(* IEC 61131-3 sources: SmartHomeNew/snapshots/clean_build_2026_04_15, 37 files *)

(* ---- E_Debug_Log_Level.dut ---- *)
{attribute 'strict'}
TYPE E_Debug_Log_Level :
(
    LOG_LEVEL_MINIMAL := 0,
    LOG_LEVEL_NORMAL := 1,
    LOG_LEVEL_VERBOSE := 2,
    LOG_LEVEL_DEBUG := 3
) USINT;
END_TYPE

(* ---- E_Zone_Access_Level.dut ---- *)
{attribute 'strict'}
TYPE E_Zone_Access_Level :
(
    ZONE_ACCESS_NONE := 0,
    ZONE_ACCESS_VIEW := 1,
    ZONE_ACCESS_CONTROL := 2,
    ZONE_ACCESS_CONFIG := 3,
    ZONE_ACCESS_FULL := 4
) USINT;
END_TYPE

(* ---- ST_BlackBox_Snapshot_V2.dut ---- *)
TYPE ST_BlackBox_Snapshot_V2 : STRUCT
    Gas_Alarm : BOOL;
    Fire_Alarm : BOOL;
    Flood_Alarm : BOOL;
    First_Fault_Type : BYTE;
    First_Fault_Source : BYTE;
END_STRUCT
END_TYPE

(* ---- ST_Boiler_Status.dut ---- *)
{attribute 'pack_mode' := '1'}
TYPE ST_Boiler_Status :
STRUCT
    Active : BOOL;
    Running : BOOL;
    Warning : BOOL;
    Error : BOOL;
    Error_ID : WORD;
    Power_Percent : REAL;
    Current_Power : REAL;
    Work_Seconds : UDINT;
    Work_Hours : REAL;
    Resource_Percent : REAL := 100.0;
    Last_Start : DT;
END_STRUCT
END_TYPE

(* ---- ST_Component_Maintenance.dut ---- *)
{attribute 'pack_mode' := '1'}
TYPE ST_Component_Maintenance :
STRUCT
    Is_Faulty : BOOL;
    Is_In_Maintenance : BOOL;
    Fallback_Value : REAL;
    Use_Last_Good_Value : BOOL;
END_STRUCT
END_TYPE

(* ---- ST_History_Event_V2.dut ---- *)
TYPE ST_History_Event_V2 : STRUCT
    Event_Code : UINT;
    Event_Value : REAL;
END_STRUCT
END_TYPE

(* ---- ST_Outdoor_Zone_Config.dut ---- *)
{attribute 'pack_mode' := '1'}
TYPE ST_Outdoor_Zone_Config :
STRUCT
    zone_id : BYTE := 0;
    lighting_circuit_id : BYTE := 0;
    auto_enabled : BOOL := TRUE;
    party_mode_enabled : BOOL := FALSE;
END_STRUCT
END_TYPE

(* ---- ST_Rule_Action.dut ---- *)
{attribute 'pack_mode' := '1'}
TYPE ST_Rule_Action :
STRUCT
    Active : BOOL;
    Triggered : BOOL;
    Action_Type : E_Rule_Action_Type;
    Target_ID : BYTE;
    Value : REAL;
END_STRUCT
END_TYPE

(* ---- ST_Valve_Test_Config.dut ---- *)
{attribute 'pack_mode' := '1'}
TYPE ST_Valve_Test_Config :
STRUCT
    valve_id : BYTE := 0;
    test_interval_days : UDINT := 7;
    Nominal_Current : REAL := 0.5;
    nominal_close_time_sec : REAL := 10.0;
    enabled : BOOL := TRUE;
END_STRUCT
END_TYPE

(* ---- GVL_COMMAND.gvl ---- *)
{attribute 'qualified_only'}
VAR_GLOBAL
    G_Gas_Valve_Close : BOOL := FALSE; // Команда: Закрыть газовый клапан
    G_Boiler_Stop : BOOL := FALSE; // Команда: Остановка котлов
    G_Supply_100_Req : BOOL := FALSE; // Команда: Приток 100%
    G_Supply_80_Req : BOOL := FALSE; // Команда: Приток 80%
    G_Vent_PV3_Boost : BOOL := FALSE; // Команда: Форсированный режим ПВ-3
    G_Exhaust_100_Req : BOOL := FALSE; // Команда: Вытяжка 100%
    G_Vent_Stop : BOOL := FALSE; // Команда: Остановка вентиляции
    G_Close_Valve_35 : BOOL := FALSE; // Команда: Закрыть вводной кран 1
    G_Close_Valve_36 : BOOL := FALSE; // Команда: Закрыть вводной кран 2
    G_Gate_Open : BOOL;
    G_Wicket_Open : BOOL;
    G_Lock_1_Open : BOOL;
    G_Lock_1_Close : BOOL;
    G_Lock_2_Open : BOOL;
    G_Lock_2_Close : BOOL;
    G_Reset_Errors : BOOL := FALSE; // Команда: Сброс ошибок
    G_Scenario_Request : E_SCENARIO_TYPE := E_SCENARIO_TYPE.SCENARIO_NONE; // Запрос на активацию сценария

    // Команды от шлюза
    G_Arm_Req : BOOL;
    G_Disarm_Req : BOOL;
    G_PIN_Code : STRING(4);
    G_RFID_Tag : STRING(20);
    G_2FA_Code_In : STRING(6);
    G_Send_2FA_Req : BOOL;
    G_2FA_Code_Out : STRING(6);
    G_Lighting_Override : ARRAY[1..32] OF BYTE;
    G_Blinds_Override : ARRAY[1..GVL_CONSTANTS.C_MAX_BLINDS] OF BYTE;
    G_Socket_Override : ARRAY[1..GVL_CONSTANTS.C_MAX_SOCKETS] OF BOOL;
    CMD_Set_Manifold_Pump_In_Service : ARRAY[1..GVL_CONSTANTS.C_MAX_MANIFOLDS] OF BOOL;
    CMD_Set_DHW_Heating_Pump_In_Service : BOOL;
    CMD_Set_DHW_Circ_Pump_In_Service : BOOL;
    CMD_Dangerous_Action_Confirm : BOOL;
    CMD_Dangerous_Action_Request : BOOL;
    CMD_User_Access_Level : INT := 0;
    CMD_Valve_Test_Open : BOOL;
    CMD_Valve_Test_Close : BOOL;
    CMD_Valve_Test_Confirm : BOOL;
    CMD_Water_Valve_Test_Open : BOOL;
    CMD_Water_Valve_Test_Close : BOOL;
    CMD_Water_Valve_Test_Confirm : BOOL;
    CMD_Gas_Valve_Test_Open : BOOL;
    CMD_Gas_Valve_Test_Close : BOOL;
    CMD_Gas_Valve_Test_Confirm : BOOL;
    CMD_Water_Selective_Recover : BOOL;
    CMD_Gas_Selective_Recover : BOOL;
END_VAR

(* ---- GVL_CONSTANTS.gvl ---- *)
{attribute 'qualified_only'}
VAR_GLOBAL CONSTANT
    // Размеры массивов (конфигурация системы)
    C_MAX_ZONES            : INT := 16; // Максимальное количество зон (комнат)
    C_MAX_LIGHTING_ZONES   : INT := 32; // Алиас для контуров освещения
    C_MAX_HEATING_CIRCUITS : INT := 8;  // Алиас для контуров отопления
    C_MAX_CLIMATE_ZONES    : INT := 16; // Алиас для климатических зон
    C_MAX_LIGHT_ZONES      : INT := 32; // Алиас для световых зон
    C_MAX_SOCKETS          : INT := 36; // Максимальное количество управляемых розеток
    C_MAX_BLINDS           : INT := 20; // Максимальное количество штор/жалюзи
    C_MAX_ALARMS           : INT := 20; // Максимальное количество активных тревог
    C_MAX_RULES            : INT := 20; // Максимальное количество правил (движок правил)
    C_MAX_MANIFOLDS        : INT := 5;  // Максимальное количество коллекторов
    C_MAX_BOILERS          : INT := 2;  // Максимальное количество котлов
    C_MAX_SUPPLY_FANS      : INT := 3;  // Максимальное количество приточных вентиляторов
    C_MAX_EXHAUST_FANS     : INT := 5;  // Максимальное количество вытяжных вентиляторов
    C_MAX_SECURITY_SENSORS : INT := 15; // Максимальное количество датчиков безопасности (герконы, стекло)
    C_MAX_FLOOD_SENSORS    : INT := 12; // Максимальное количество датчиков протечки
    C_MAX_DOOR_SENSORS     : INT := 8;  // Максимальное количество датчиков дверей
    C_MAX_CO_SENSORS       : INT := 8;  // Максимальное количество датчиков CO
    C_MAX_METHANE_SENSORS  : INT := 2;  // Максимальное количество датчиков метана
    C_MAX_VENT_UNITS       : INT := 8;  // Максимальное количество вентустановок
    C_MAX_SUPPLY_TEMPS     : INT := 2;  // Максимальное количество датчиков температуры притока
    C_MAX_SMOKE_SENSORS    : INT := 6;  // Максимальное количество датчиков дыма
    C_MAX_SCENARIOS        : INT := 6;  // Максимальное количество сценариев
    C_MAX_OUTDOOR_ZONES    : INT := 4;  // Максимальное количество зон уличного освещения
    C_MAX_ACCESS_CODES     : INT := 10; // Максимальное количество кодов доступа
    C_MAX_WET_ZONES        : INT := 4;  // Максимальное количество "мокрых" зон (санузлы)
    C_MAX_CALIBRATIONS     : INT := 20; // Максимальное количество калибровок датчиков
    C_MAX_MODULES          : INT := 10; // Максимальное количество модулей ввода-вывода
    C_MAX_CLEANING_MODES   : INT := 3;  // Максимальное количество режимов уборки
    C_MAX_ALLOWED_IPS      : INT := 5;  // Максимальное количество разрешенных IP-адресов
    C_MAX_VENT_SUPPLY_MODES: INT := 3;  // Максимальное количество режимов притока вентиляции
    C_MAX_SECURITY_PHONES  : INT := 5;  // Максимальное количество телефонов для оповещения
    C_MAX_FLOOD_VALVES     : INT := 3;  // Максимальное количество кранов защиты от протечек
    C_MAX_HUMIDITY_SENSORS : INT := 8;  // Максимальное количество датчиков влажности
    C_MAX_CO2_SENSORS      : INT := 8;  // Максимальное количество датчиков CO2
    C_MAX_CIRCUITS_PER_MANIFOLD : INT := 4; // Максимальное количество контуров на коллектор
    C_MAX_TREND_DATA_POINTS: INT := 100; // Максимальное количество точек данных для трендов
    C_MAX_HISTORY_RECORDS  : INT := 100; // Максимальное количество записей в истории
    C_MAX_DEBUG_LOGS       : INT := 1000; // Максимальное количество записей в логе отладки
    C_MAX_GATEWAY_COMMANDS : INT := 10; // Максимальное количество команд в буфере шлюза
    C_MAX_STATE_SNAPSHOTS  : INT := 10; // Максимальное количество снимков состояния
    C_MAX_BLACKBOX_RECORDS : INT := 100; // Максимальное количество записей черного ящика
    C_MAX_PRESENCE_HISTORY : INT := 1008; // Максимальное количество записей истории присутствия
    C_MAX_MODBUS_REGISTERS : INT := 201; // Максимальное количество регистров Modbus
    C_MAX_DEDUPLICATION_HISTORY : INT := 100; // Максимальное количество записей истории дедупликации
    C_MAX_NVRAM_RECORDS    : INT := 100; // Максимальное количество записей NVRAM
    C_MAX_NVRAM_DATA       : INT := 128; // Максимальный размер данных NVRAM

    // Аналоговые входы (4-20mA, 0-10V)
    C_ANALOG_RAW_MAX       : WORD := 27648; // Максимальное значение АЦП (100%)
    C_ANALOG_4MA_RAW       : WORD := 5529;  // Значение АЦП для 4mA (20% от 27648)
    C_ANALOG_3_6MA_RAW     : WORD := 4976;  // Порог обрыва NAMUR NE43 (< 3.6mA)
    C_ANALOG_21MA_RAW      : WORD := 29030; // Порог КЗ NAMUR NE43 (> 21mA)
    C_ANALOG_10V_MAX_RAW   : WORD := 30000; // Порог выхода за пределы 0-10V

    // Временные константы (в миллисекундах)
    C_MS_IN_SECOND         : UDINT := 1000;
    C_MS_IN_MINUTE         : UDINT := 60000;
    C_MS_IN_HOUR           : UDINT := 3600000;
    C_MS_IN_DAY            : UDINT := 86400000;

    // Пороги мощности для каскада котлов (0..500%)
    C_BOILER_CASCADE_MIN_DEMAND : REAL := 25.0; // Минимальный запрос для включения ведущего котла (5% от одного коллектора)
    C_BOILER_CASCADE_HIGH_DEMAND : REAL := 250.0; // Высокий запрос для включения второго котла (50% от общей мощности)
END_VAR

(* ---- GVL_GATEWAY.gvl ---- *)
{attribute 'qualified_only'}
VAR_GLOBAL
    G_Gateway_Command : ST_Gateway_Command;
    G_Gateway_Command_Received : BOOL;
    G_Gateway_Send_2FA : BOOL;
    G_Gateway_2FA_Code : STRING(6);
    G_Gateway_Telegram_Msg : STRING(200);
    G_Gateway_Send_Telegram : BOOL;
    G_Gateway_HMI_Status_Message : STRING(200);
    G_Gateway_Ping_OK : BOOL;
    G_Gateway_Data_Ready : BOOL;
    G_Gateway_Modbus_Registers : ARRAY[0..GVL_CONSTANTS.C_MAX_MODBUS_REGISTERS-1] OF WORD;
END_VAR

(* ---- GVL_STATE.gvl ---- *)
{attribute 'qualified_only'}
VAR_GLOBAL
    G_Floor_Temps : ARRAY[1..8] OF REAL; // Массив текущих температур поверхности пола
    G_Room_Temps : ARRAY[1..GVL_CONSTANTS.C_MAX_ZONES] OF REAL;
    G_Room_Hum : ARRAY[1..GVL_CONSTANTS.C_MAX_ZONES] OF REAL;
    G_Room_CO2 : ARRAY[1..GVL_CONSTANTS.C_MAX_ZONES] OF REAL;
    G_Motion_Sensors : ARRAY[1..32] OF BOOL;
    G_Door_Sensors : ARRAY[1..GVL_CONSTANTS.C_MAX_DOOR_SENSORS] OF BOOL;
    G_Window_Sensors : ARRAY[1..GVL_CONSTANTS.C_MAX_ZONES] OF BOOL;
    G_Water_Sensors : ARRAY[1..GVL_CONSTANTS.C_MAX_FLOOD_SENSORS] OF BOOL;
    G_Smoke_Sensors : ARRAY[1..GVL_CONSTANTS.C_MAX_SMOKE_SENSORS] OF BOOL;
    G_Methane_Sensors : ARRAY[1..GVL_CONSTANTS.C_MAX_METHANE_SENSORS] OF REAL;
    G_CO_Sensors : ARRAY[1..GVL_CONSTANTS.C_MAX_CO_SENSORS] OF REAL;
    G_Manifold_Pressures : ARRAY[1..GVL_CONSTANTS.C_MAX_MANIFOLDS] OF REAL;
    G_Manifold_Currents : ARRAY[1..GVL_CONSTANTS.C_MAX_MANIFOLDS] OF REAL;
    G_Manifold_T_Supply : ARRAY[1..GVL_CONSTANTS.C_MAX_MANIFOLDS] OF REAL;
    G_Manifold_T_Return : ARRAY[1..GVL_CONSTANTS.C_MAX_MANIFOLDS] OF REAL;
    G_Boiler_Flame : ARRAY[1..GVL_CONSTANTS.C_MAX_BOILERS] OF BOOL;
    G_Boiler_Error : ARRAY[1..GVL_CONSTANTS.C_MAX_BOILERS] OF BOOL;
    G_Boiler_OT_Online : ARRAY[1..GVL_CONSTANTS.C_MAX_BOILERS] OF BOOL; // Статус доступности OpenTherm-канала котла от реального OT-адаптера/драйвера
    G_Boiler_OT_Enable : ARRAY[1..GVL_CONSTANTS.C_MAX_BOILERS] OF BOOL; // Команды разрешения через OpenTherm
    G_Boiler_OT_Setpoint : ARRAY[1..GVL_CONSTANTS.C_MAX_BOILERS] OF REAL; // Уставки через OpenTherm
    G_Physical_Switches : ARRAY[1..32] OF BOOL;
    G_Socket_Switches : ARRAY[1..GVL_CONSTANTS.C_MAX_SOCKETS] OF BOOL; // Legacy-поле: локальные выключатели розеток не используются
    G_Outdoor_Temp : REAL;
    G_Supply_Temps : ARRAY[1..GVL_CONSTANTS.C_MAX_SUPPLY_TEMPS] OF REAL; // Температура приточного воздуха после калорифера
    G_DHW_Temp : REAL;
    G_DHW_Pressure : REAL;
    G_Zone_Valves : ARRAY[1..8] OF BOOL;
    G_Manifold_Pumps : ARRAY[1..GVL_CONSTANTS.C_MAX_MANIFOLDS] OF BOOL;
    G_Manifold_Valves : ARRAY[1..GVL_CONSTANTS.C_MAX_MANIFOLDS] OF REAL; // 0.0 - 1.0
    G_Manifold_End_Switches : ARRAY[1..GVL_CONSTANTS.C_MAX_MANIFOLDS] OF BOOL; // Концевики клапанов
    G_Supply_Fans : ARRAY[1..GVL_CONSTANTS.C_MAX_SUPPLY_FANS] OF REAL; // 0.0 - 1.0
    G_Exhaust_Fans : ARRAY[1..GVL_CONSTANTS.C_MAX_EXHAUST_FANS] OF REAL; // 0.0 - 1.0
    G_Vent_Heater_Power : ARRAY[1..GVL_CONSTANTS.C_MAX_BOILERS] OF REAL;
    G_Lighting_Levels : ARRAY[1..32] OF BYTE;
    G_Blinds_Positions : ARRAY[1..GVL_CONSTANTS.C_MAX_BLINDS] OF BYTE;
    G_Socket_States : ARRAY[1..GVL_CONSTANTS.C_MAX_SOCKETS] OF BOOL;
    G_DHW_Heating_Pump : BOOL;
    G_DHW_Circ_Pump : BOOL;
    G_Backup_Circulation_Pump : BOOL; // Резервный циркуляционный насос для антизамерзания при газовой аварии
    G_Electric_Heater_Enable : BOOL; // Сухой контакт электрического нагревателя для антизамерзания
    G_Safety_Gas_Alarm : BOOL;
    G_Safety_Leak_Alarm : BOOL;
    G_Safety_Smoke_Alarm : BOOL;
    G_Safety_Emergency_Stop : BOOL; // агрегированный аварийный стоп
    G_Safety_Gas_Latched : BOOL; // защёлкнутая газовая авария
    G_Safety_Leak_Latched : BOOL; // защёлкнутая авария протечки
    G_Safety_Smoke_Latched : BOOL; // защёлкнутая дымовая/пожарная авария
    G_Safety_Freeze_Risk : BOOL; // риск замерзания при защёлкнутой газовой аварии
    G_System_Mode : E_System_Operating_Mode := E_System_Operating_Mode.MODE_NORMAL; // Текущий режим работы системы
    G_System_Mode_Text : STRING(64);
    G_Heating_IO_Fault : BOOL;
    G_Heating_Sensor_Fault : BOOL;
    G_Heating_Subsystem_Degraded : BOOL;
    G_DHW_IO_Fault : BOOL;
    G_DHW_Sensor_Fault : BOOL;
    G_DHW_Subsystem_Degraded : BOOL;
    G_Ventilation_IO_Fault : BOOL;
    G_Ventilation_Subsystem_Degraded : BOOL;
    G_Lighting_IO_Fault : BOOL;
    G_Lighting_Subsystem_Degraded : BOOL;
    G_Access_Comm_Fault : BOOL;
    G_Evacuation_Lighting_Active : BOOL;
    G_Evac_Hazard_Zone : ARRAY[1..32] OF BOOL; // опасные зоны (дым/протечка)
    G_Evac_Guidance : ARRAY[1..32] OF INT; // -1 = избегать, 0 = нейтрально, +1 = к выходу
 // Активен режим световой эвакуации // Текстовый статус режима работы системы

    G_Rule_Actions : ARRAY[1..GVL_CONSTANTS.C_MAX_RULES] OF ST_Rule_Action;
    G_Sim_Lights : ARRAY[1..32] OF BOOL;
    G_Freeze_Hardware_Degraded : BOOL; // Деградация anti-freeze hardware
    G_Freeze_Hardware_Failed : BOOL; // Критический отказ anti-freeze hardware
    G_Water_Zone_Enable : ARRAY[1..32] OF BOOL; // Селективное открытие воды по зонам
    G_Water_Zone_Open_FB : ARRAY[1..32] OF BOOL; // Обратная связь: зональный клапан открыт
    G_Water_Zone_Close_FB : ARRAY[1..32] OF BOOL; // Обратная связь: зональный клапан закрыт
    G_Water_Zone_Exercise_Active : ARRAY[1..32] OF BOOL; // Профилактическая прокрутка шаровых кранов
END_VAR

(* ---- FB_Alarm_V2_Core.st ---- *)
FUNCTION_BLOCK FB_Alarm_V2_Core
VAR_INPUT
    VI_System_Time_MS : UDINT;
    VI_Pending_Alarms : ARRAY[1..10] OF ST_Alarm_Record;
END_VAR
VAR_IN_OUT
    VIO_Alarm_List : ARRAY[1..GVL_CONSTANTS.C_MAX_ALARMS] OF ST_Alarm_Record;
    VIO_Next_Alarm_ID : UDINT;
END_VAR
VAR_OUTPUT
    VO_Event_Pulse : BOOL;
    VO_Event_Code : UDINT;
    VO_Event_Value : REAL;
END_VAR

VO_Event_Pulse := FALSE;
VO_Event_Code := 0;
VO_Event_Value := 0.0;
END_FUNCTION_BLOCK

(* ---- FB_BlackBox_Recorder.st ---- *)
FUNCTION_BLOCK FB_BlackBox_Recorder
VAR_INPUT
    VI_Current_Data : ST_BlackBox_Record;
    VI_Freeze       : BOOL;
END_VAR
VAR_OUTPUT
    VO_Frozen       : BOOL;
    VO_Records_Count: INT;
END_VAR
VAR
    L_Write_Index   : INT := 0;
    L_Initialized   : BOOL := FALSE;
END_VAR

IF NOT L_Initialized THEN
    L_Write_Index := GVL_Retain.G_BlackBox_LastIndex;
    IF L_Write_Index < 0 OR L_Write_Index >= GVL_CONSTANTS.C_MAX_BLACKBOX_RECORDS THEN
        L_Write_Index := 0;
        GVL_Retain.G_BlackBox_LastIndex := 0;
    END_IF;
    L_Initialized := TRUE;
END_IF;

IF VI_Freeze THEN
    GVL_Retain.G_BlackBox_Frozen := TRUE;
END_IF;

VO_Frozen := GVL_Retain.G_BlackBox_Frozen;

IF NOT GVL_Retain.G_BlackBox_Frozen THEN
    GVL_Retain.G_BlackBox_Buffer[L_Write_Index] := VI_Current_Data;
    GVL_Retain.G_BlackBox_LastIndex := L_Write_Index;

    L_Write_Index := L_Write_Index + 1;
    IF L_Write_Index >= GVL_CONSTANTS.C_MAX_BLACKBOX_RECORDS THEN
        L_Write_Index := 0;
    END_IF;
END_IF;

VO_Records_Count := GVL_CONSTANTS.C_MAX_BLACKBOX_RECORDS; // Размер кольцевого буфера
// >>> BULK_SYNC_ANCHOR: FB_BlackBox_Recorder <<<

(* ---- FB_Boiler_Cascade_Manager.st ---- *)
FUNCTION_BLOCK FB_Boiler_Cascade_Manager
VAR_INPUT
    VI_Enable : BOOL;
    VI_System_Time_MS : UDINT;
    VI_Boiler_Stop : BOOL;

    VI_DHW_Heating_Demand : BOOL;
    VI_DHW_Target_Temp : REAL;

    VI_Target_Supply_Temp : REAL;
    VI_Demand_Power : REAL; // 0..500% (сумма запросов от 5 смесительных узлов)

    VI_Boiler_Flame_Status : ARRAY[1..GVL_CONSTANTS.C_MAX_BOILERS] OF BOOL;
    VI_Boiler_Error_Status : ARRAY[1..GVL_CONSTANTS.C_MAX_BOILERS] OF BOOL;
    VI_Boiler_OT_Online : ARRAY[1..GVL_CONSTANTS.C_MAX_BOILERS] OF BOOL;
    VI_Boiler_Modulation : ARRAY[1..GVL_CONSTANTS.C_MAX_BOILERS] OF REAL;
END_VAR

VAR_OUTPUT
    VO_Boiler_Enable : ARRAY[1..GVL_CONSTANTS.C_MAX_BOILERS] OF BOOL;
    VO_Boiler_Setpoint : ARRAY[1..GVL_CONSTANTS.C_MAX_BOILERS] OF REAL;
    VO_Lead_Boiler : BYTE;
END_VAR

VAR
    L_i : INT;
    L_Lead_Boiler : BYTE := 1;

    L_Last_Rotation_MS : UDINT := 0;
    L_Rotation_Initialized : BOOL := FALSE;
    L_Rotation_Period_MS : UDINT := 604800000; // 168h

    L_Lead_Available : BOOL;
    L_Reserve_Available : BOOL;
    L_Reserve_Boiler : BYTE;
    L_Start_Reserve : BOOL;
    L_Target_Setpoint : REAL;
    L_Flame_Miss_Timer : ARRAY[1..GVL_CONSTANTS.C_MAX_BOILERS] OF TON;
END_VAR

// Сброс выходов по умолчанию
FOR L_i := 1 TO GVL_CONSTANTS.C_MAX_BOILERS DO
    VO_Boiler_Enable[L_i] := FALSE;
    VO_Boiler_Setpoint[L_i] := 0.0;
END_FOR;

// Инициализация ротации
IF NOT L_Rotation_Initialized THEN
    L_Last_Rotation_MS := VI_System_Time_MS;
    L_Rotation_Initialized := TRUE;
END_IF;

// Принудительная остановка
IF VI_Boiler_Stop THEN
    VO_Lead_Boiler := L_Lead_Boiler;
    RETURN;
END_IF;

// Ротация строго каждые 168 часов
IF (VI_System_Time_MS - L_Last_Rotation_MS) >= L_Rotation_Period_MS THEN
    IF GVL_CONSTANTS.C_MAX_BOILERS > 1 THEN
        L_Lead_Boiler := 3 - L_Lead_Boiler;
    END_IF;
    L_Last_Rotation_MS := VI_System_Time_MS;
END_IF;

L_Reserve_Boiler := SEL(L_Lead_Boiler = 1, 1, 2);

L_Lead_Available :=
    VI_Boiler_OT_Online[L_Lead_Boiler] AND
    NOT VI_Boiler_Error_Status[L_Lead_Boiler];

L_Reserve_Available :=
    (GVL_CONSTANTS.C_MAX_BOILERS > 1) AND
    VI_Boiler_OT_Online[L_Reserve_Boiler] AND
    NOT VI_Boiler_Error_Status[L_Reserve_Boiler];

// Контроль "команда есть, пламени нет" для ведущего котла
L_Flame_Miss_Timer[L_Lead_Boiler](
    IN := VI_Enable AND L_Lead_Available AND NOT VI_DHW_Heating_Demand AND NOT VI_Boiler_Flame_Status[L_Lead_Boiler],
    PT := T#120s
);

IF L_Flame_Miss_Timer[L_Lead_Boiler].Q AND L_Reserve_Available THEN
    L_Lead_Boiler := L_Reserve_Boiler;
    L_Last_Rotation_MS := VI_System_Time_MS;
    L_Lead_Available :=
        VI_Boiler_OT_Online[L_Lead_Boiler] AND
        NOT VI_Boiler_Error_Status[L_Lead_Boiler];
    L_Reserve_Boiler := SEL(L_Lead_Boiler = 1, 1, 2);
    L_Reserve_Available :=
        (GVL_CONSTANTS.C_MAX_BOILERS > 1) AND
        VI_Boiler_OT_Online[L_Reserve_Boiler] AND
        NOT VI_Boiler_Error_Status[L_Reserve_Boiler];
END_IF;

// Нет запроса тепла
IF NOT VI_Enable THEN
    VO_Lead_Boiler := L_Lead_Boiler;
    RETURN;
END_IF;

// Целевая уставка
IF VI_DHW_Heating_Demand THEN
    L_Target_Setpoint := LIMIT(20.0, VI_DHW_Target_Temp + 15.0, 85.0);
ELSE
    L_Target_Setpoint := LIMIT(20.0, VI_Target_Supply_Temp + 5.0, 80.0);
END_IF;

// Выбор ведущего по доступности
IF NOT L_Lead_Available AND L_Reserve_Available THEN
    L_Lead_Boiler := L_Reserve_Boiler;
    L_Lead_Available := TRUE;
    L_Reserve_Boiler := SEL(L_Lead_Boiler = 1, 1, 2);
    L_Reserve_Available :=
        (GVL_CONSTANTS.C_MAX_BOILERS > 1) AND
        VI_Boiler_OT_Online[L_Reserve_Boiler] AND
        NOT VI_Boiler_Error_Status[L_Reserve_Boiler];
END_IF;

// Основной котёл
IF L_Lead_Available THEN
    VO_Boiler_Enable[L_Lead_Boiler] := TRUE;
    VO_Boiler_Setpoint[L_Lead_Boiler] := L_Target_Setpoint;
END_IF;

// Резервный котёл: >80% или отказ основного
L_Start_Reserve :=
    L_Reserve_Available AND
    (
        (VI_Demand_Power > 80.0) OR
        (NOT L_Lead_Available)
    );

IF L_Start_Reserve THEN
    VO_Boiler_Enable[L_Reserve_Boiler] := TRUE;
    VO_Boiler_Setpoint[L_Reserve_Boiler] := L_Target_Setpoint;
END_IF;

VO_Lead_Boiler := L_Lead_Boiler;

(* ---- FB_Emergency_Valve_Open.st ---- *)
FUNCTION_BLOCK FB_Emergency_Valve_Open
VAR_INPUT
    VI_Fire_Alarm : BOOL; // Сигнал пожарной тревоги
    VI_Gas_Alarm  : BOOL; // Сигнал газовой тревоги
END_VAR
VAR_OUTPUT
    VO_Open_Cmd   : BOOL; // Команда на аварийное открытие клапана
END_VAR

// Приоритетное открытие при любой серьезной аварии
VO_Open_Cmd := VI_Fire_Alarm OR VI_Gas_Alarm;

(* ---- FB_FloorHeating_Freeze_Protection.st ---- *)
FUNCTION_BLOCK FB_FloorHeating_Freeze_Protection
VAR_INPUT
    VI_Outdoor_Temp : REAL;
    VI_Threshold : REAL := 7.0;
END_VAR
VAR_IN_OUT
    VI_Floor_Temps : ARRAY[1..GVL_CONSTANTS.C_MAX_HEATING_CIRCUITS] OF REAL;
END_VAR
VAR_OUTPUT
    VO_Freeze_Alert : BOOL;
    VO_Pump_Force_On : BOOL;
END_VAR
VAR
    L_i : INT;
END_VAR

VO_Freeze_Alert := FALSE;
VO_Pump_Force_On := FALSE;

FOR L_i := 1 TO GVL_CONSTANTS.C_MAX_HEATING_CIRCUITS DO
    IF VI_Floor_Temps[L_i] < VI_Threshold THEN
        VO_Freeze_Alert := TRUE;
        VO_Pump_Force_On := TRUE;
        RETURN;
    END_IF;
END_FOR;

IF VI_Outdoor_Temp < -5.0 THEN
    VO_Pump_Force_On := TRUE;
END_IF;

(* ---- FB_FloorHeating_Overheat_Protection.st ---- *)
FUNCTION_BLOCK FB_FloorHeating_Overheat_Protection
VAR_INPUT
    VI_Threshold : REAL := 45.0;
END_VAR
VAR_IN_OUT
    VI_Temps : ARRAY[1..GVL_CONSTANTS.C_MAX_HEATING_CIRCUITS] OF REAL;
END_VAR
VAR_OUTPUT
    VO_Overheat_Detected : BOOL;
    VO_Locked_Circuits : ARRAY[1..GVL_CONSTANTS.C_MAX_HEATING_CIRCUITS] OF BOOL;
END_VAR
VAR
    L_i : INT;
END_VAR

VO_Overheat_Detected := FALSE;
FOR L_i := 1 TO GVL_CONSTANTS.C_MAX_HEATING_CIRCUITS DO
    IF VI_Temps[L_i] > VI_Threshold THEN
        VO_Overheat_Detected := TRUE;
        VO_Locked_Circuits[L_i] := TRUE;
    END_IF;
END_FOR;

(* ---- FB_IO_Module_Watchdog.st ---- *)
FUNCTION_BLOCK FB_IO_Module_Watchdog
VAR_INPUT
    VI_System_Time_MS : UDINT;
    VI_Module_ID : BYTE;
    VI_Heartbeat_Signal : BOOL; // Сигнал от модуля (например, мигающий бит)
    VI_Timeout_MS : UDINT := 2000; // Таймаут 2 секунды по умолчанию
END_VAR
VAR_OUTPUT
    VO_Module_Online : BOOL;
    VO_Error_Active : BOOL;
END_VAR
VAR
    L_Last_Heartbeat_State : BOOL;
    L_Last_Heartbeat_Time : UDINT;
    L_Elapsed_Time : UDINT;
END_VAR

// Отслеживание изменения сигнала
IF VI_Heartbeat_Signal <> L_Last_Heartbeat_State THEN
    L_Last_Heartbeat_Time := VI_System_Time_MS;
    L_Last_Heartbeat_State := VI_Heartbeat_Signal;
END_IF;

// Проверка таймаута
L_Elapsed_Time := (SEL(VI_System_Time_MS >= L_Last_Heartbeat_Time, VI_System_Time_MS - L_Last_Heartbeat_Time, (4294967295 - L_Last_Heartbeat_Time) + VI_System_Time_MS + 1));

IF L_Elapsed_Time > VI_Timeout_MS THEN
    VO_Module_Online := FALSE;
    VO_Error_Active := TRUE;
ELSE
    VO_Module_Online := TRUE;
    VO_Error_Active := FALSE;
END_IF;
// >>> BULK_SYNC_ANCHOR: FB_IO_Module_Watchdog <<<

(* ---- FB_Lighting_Blinds_Manager.st ---- *)
FUNCTION_BLOCK FB_Lighting_Blinds_Manager
// Менеджер управления освещением и шторами/жалюзи.
// Обеспечивает работу по сценариями, датчикам движения, физическим выключателям и правилам.
VAR_INPUT
    VI_System_Time_MS : UDINT; // Системное время в миллисекундах
    VI_IsActivePLC : BOOL; // Флаг активности ПЛК (TRUE = ведущий)
    VI_Current_Scenario : E_SCENARIO_TYPE; // Текущий глобальный сценарий (Утро, Вечер, Сон, Никого нет)
    VI_Away_Level : BYTE; // Уровень режима "Никого нет" (1-Короткий, 2-Средний, 3-Длительный)
    VI_Simulation_Active : BOOL; // Флаг активности симуляции присутствия
    VI_Is_Night : BOOL; // Флаг ночного времени (по астрономическому таймеру)
    VI_System_Mode : E_System_Operating_Mode; // Агрегированный режим работы системы
END_VAR
VAR_IN_OUT
    VI_Manual_Light_Override : ARRAY[1..32] OF BYTE; // Ручное переопределение яркости (0-100%)
    VI_Manual_Blinds_Override : ARRAY[1..GVL_CONSTANTS.C_MAX_BLINDS] OF BYTE; // Ручное переопределение позиции штор (0-100%)
    VI_Simulation_Lights : ARRAY[1..32] OF BOOL; // Состояния света от симулятора
    VI_Physical_Switches : ARRAY[1..32] OF BOOL; // Состояния физических выключателей
    VI_Motion_Sensors : ARRAY[1..32] OF BOOL; // Состояния датчиков движения
    VI_Rule_Actions : ARRAY[1..GVL_CONSTANTS.C_MAX_RULES] OF ST_Rule_Action; // Действия от Rule Engine
    VI_IO_Modules_Online : ARRAY[1..GVL_CONSTANTS.C_MAX_MODULES] OF BOOL; // Статусы модулей ввода-вывода
    VI_Wet_Zone_Map : ARRAY[1..32] OF BOOL; // Карта мокрых зон
    VI_Scenario_Configs : ARRAY[1..GVL_CONSTANTS.C_MAX_SCENARIOS] OF ST_Scenario_Config; // Конфигурации сценариев
END_VAR
VAR_OUTPUT
    VO_Lighting_Levels : ARRAY[1..32] OF BYTE; // Выходные уровни освещения (0-100%)
    VO_Blinds_Positions : ARRAY[1..GVL_CONSTANTS.C_MAX_BLINDS] OF BYTE; // Выходные позиции штор (0-100%)
    VO_Wet_Zone_Light_Active : ARRAY[1..GVL_CONSTANTS.C_MAX_WET_ZONES] OF BOOL; // Флаги включенного света в мокрых зонах (для вентиляции)
END_VAR
VAR
    // Blinds V2 shadow (phase2)
    fbBlindsV2Staging : FB_Blinds_V2_Staging;
    L_Blinds_V2_Command_Shadow : ST_Blinds_Command_V2;
    L_Blinds_V2_State_Shadow : ST_Blinds_State_V2;
    L_Blinds_V2_Shadow_Diff_Found : BOOL;
    L_Blinds_V2_Switch_Enabled : BOOL;
    L_Blinds_V2_Path_Ready : BOOL;
    L_Blinds_Using_Legacy_Fallback : BOOL;
    // Lighting V2 shadow (phase2)
    fbLightingV2Staging : FB_Lighting_V2_Staging;
    L_Lighting_V2_Command_Shadow : ST_Lighting_Command_V2;
    L_Lighting_V2_State_Shadow : ST_Lighting_State_V2;
    L_Lighting_V2_Shadow_Diff_Found : BOOL;
    L_Lighting_V2_Switch_Enabled : BOOL;
    L_Lighting_V2_Path_Ready : BOOL;
    L_Lighting_Using_Legacy_Fallback : BOOL;
    L_i : INT;
    L_j : INT;
    L_Base_Light : BYTE;
    L_Base_Blinds : BYTE;
    L_Target_Base_Light : BYTE;
    L_Target_Base_Blinds : BYTE;
    L_Prev_Scenario : E_SCENARIO_TYPE;
    L_Transition_Light : FB_Scenario_Transition_Controller;
    L_Transition_Blinds : FB_Scenario_Transition_Controller;
    L_Light_States : ARRAY[1..32] OF BOOL;
    L_Prev_Switches : ARRAY[1..32] OF BOOL;
    L_Prev_Motion_Q : ARRAY[1..32] OF BOOL;
    L_Manual_Override : ARRAY[1..32] OF BOOL; // Флаг ручного переопределения (выключателем)
    L_Motion_Timers : ARRAY[1..32] OF FB_System_Timer_TOF;
    L_Rule_Light_Active : BOOL;
    L_Rule_Light_Val : BYTE;
    L_Rule_Blinds_Active : BOOL;
    L_Rule_Blinds_Val : BYTE;
    L_Wet_Zone_Idx : INT;
    L_Effective_Scenario : E_SCENARIO_TYPE;
    L_Effective_Simulation_Active : BOOL;
END_VAR

IF NOT VI_IsActivePLC THEN RETURN; END_IF;

L_Lighting_V2_Shadow_Diff_Found := FALSE;
L_Blinds_V2_Shadow_Diff_Found := FALSE;
L_Blinds_V2_Switch_Enabled := TRUE;
L_Blinds_V2_Path_Ready := FALSE;
L_Blinds_Using_Legacy_Fallback := TRUE;
L_Lighting_V2_Switch_Enabled := TRUE;
L_Lighting_V2_Path_Ready := FALSE;
L_Lighting_Using_Legacy_Fallback := TRUE;

GVL_STATE.G_Lighting_IO_Fault := FALSE;
GVL_STATE.G_Lighting_Subsystem_Degraded := FALSE;

L_Effective_Scenario := VI_Current_Scenario;
L_Effective_Simulation_Active := VI_Simulation_Active;

CASE VI_System_Mode OF
    E_System_Operating_Mode.MODE_SAFE_STOP:
        FOR L_j := 1 TO 32 DO
            VO_Lighting_Levels[L_j] := 0;
        END_FOR;
        FOR L_j := 1 TO GVL_CONSTANTS.C_MAX_BLINDS DO
            VO_Blinds_Positions[L_j] := 100;
        END_FOR;
        FOR L_j := 1 TO GVL_CONSTANTS.C_MAX_WET_ZONES DO
            VO_Wet_Zone_Light_Active[L_j] := FALSE;
        END_FOR;
        RETURN;
    E_System_Operating_Mode.MODE_FREEZE_PROTECTION:
        L_Effective_Scenario := E_SCENARIO_TYPE.SCENARIO_NONE;
        L_Effective_Simulation_Active := FALSE;
    E_System_Operating_Mode.MODE_DEGRADED:
        L_Effective_Simulation_Active := FALSE;
END_CASE;

// Инициализация индекса мокрых зон
L_Wet_Zone_Idx := 1;
// Сброс массива мокрых зон
FOR L_i := 1 TO GVL_CONSTANTS.C_MAX_WET_ZONES DO
    VO_Wet_Zone_Light_Active[L_i] := FALSE;
END_FOR;

// Проверка связи с модулями ввода-вывода
FOR L_i := 1 TO GVL_CONSTANTS.C_MAX_MODULES DO
    IF NOT VI_IO_Modules_Online[L_i] THEN
        GVL_STATE.G_Lighting_IO_Fault := TRUE;
GVL_STATE.G_Lighting_Subsystem_Degraded := TRUE;
        // Переход в безопасное состояние при потере связи (свет выкл, шторы открыты для эвакуации)
        FOR L_j := 1 TO 32 DO
            VO_Lighting_Levels[L_j] := 0;
        END_FOR;
        FOR L_j := 1 TO GVL_CONSTANTS.C_MAX_BLINDS DO
            VO_Blinds_Positions[L_j] := 100;
        END_FOR;
        RETURN;
    END_IF;
END_FOR;

// 1. Определение целевых уровней по сценарию (ТЗ 7.1)
IF L_Effective_Scenario >= 1 AND L_Effective_Scenario <= GVL_CONSTANTS.C_MAX_SCENARIOS THEN
    L_Target_Base_Light := VI_Scenario_Configs[L_Effective_Scenario].lighting_level_base;
    L_Target_Base_Blinds := VI_Scenario_Configs[L_Effective_Scenario].blinds_position_percent;
ELSE
    L_Target_Base_Light := 100;
    L_Target_Base_Blinds := 100;
END_IF;

// Корректировка по астрономическому таймеру
IF VI_Is_Night AND L_Effective_Scenario <> E_SCENARIO_TYPE.SCENARIO_AWAY AND L_Effective_Scenario <> E_SCENARIO_TYPE.SCENARIO_SLEEP THEN
    L_Target_Base_Blinds := 0; // Закрывать шторы ночью
END_IF;

// Плавный переход при смене сценария
IF L_Effective_Scenario <> L_Prev_Scenario THEN
    L_Transition_Light(
        VI_System_Time := VI_System_Time_MS,
        VI_Start_Time := VI_System_Time_MS,
        VI_Duration := 5000, // 5 секунд на плавное изменение света
        VI_Start_Value := TO_REAL(L_Base_Light),
        VI_End_Value := TO_REAL(L_Target_Base_Light)
    );
    L_Transition_Blinds(
        VI_System_Time := VI_System_Time_MS,
        VI_Start_Time := VI_System_Time_MS,
        VI_Duration := 10000, // 10 секунд на плавное изменение штор
        VI_Start_Value := TO_REAL(L_Base_Blinds),
        VI_End_Value := TO_REAL(L_Target_Base_Blinds)
    );
    L_Prev_Scenario := L_Effective_Scenario;
ELSE
    L_Transition_Light(
        VI_System_Time := VI_System_Time_MS,
        VI_Start_Time := L_Transition_Light.VI_Start_Time,
        VI_Duration := L_Transition_Light.VI_Duration,
        VI_Start_Value := L_Transition_Light.VI_Start_Value,
        VI_End_Value := TO_REAL(L_Target_Base_Light)
    );
    L_Transition_Blinds(
        VI_System_Time := VI_System_Time_MS,
        VI_Start_Time := L_Transition_Blinds.VI_Start_Time,
        VI_Duration := L_Transition_Blinds.VI_Duration,
        VI_Start_Value := L_Transition_Blinds.VI_Start_Value,
        VI_End_Value := TO_REAL(L_Target_Base_Blinds)
    );
END_IF;

L_Base_Light := TO_BYTE(L_Transition_Light.VO_Current_Value);
L_Base_Blinds := TO_BYTE(L_Transition_Blinds.VO_Current_Value);

// 2. Управление освещением
FOR L_i := 1 TO 32 DO
    L_Rule_Light_Active := FALSE;
    L_Rule_Light_Val := 0;

    // Проверка правил
    FOR L_j := 1 TO GVL_CONSTANTS.C_MAX_RULES DO
        IF VI_Rule_Actions[L_j].Active AND VI_Rule_Actions[L_j].Target_ID = L_i THEN
            IF VI_Rule_Actions[L_j].Action_Type = E_Rule_Action_Type.ACTION_SET_LIGHTING_BASE THEN
                L_Rule_Light_Active := TRUE;
                L_Rule_Light_Val := REAL_TO_BYTE(VI_Rule_Actions[L_j].Value);
                L_Light_States[L_i] := (L_Rule_Light_Val > 0);
            ELSIF VI_Rule_Actions[L_j].Action_Type = E_Rule_Action_Type.ACTION_TOGGLE_LIGHTING AND VI_Rule_Actions[L_j].Triggered THEN
                L_Light_States[L_i] := NOT L_Light_States[L_i];
            END_IF;
        END_IF;
    END_FOR;

    // Приоритет 1: Физические выключатели (ТЗ 1.0)
    IF VI_Physical_Switches[L_i] AND NOT L_Prev_Switches[L_i] THEN
        L_Light_States[L_i] := NOT L_Light_States[L_i];
        L_Manual_Override[L_i] := TRUE; // Запоминаем ручное переопределение
    END_IF;
    L_Prev_Switches[L_i] := VI_Physical_Switches[L_i];

    // Приоритет 2: Датчики движения (ТЗ 2.0)
    // Защита от дребезга и удержание сигнала движения с помощью TOF
    L_Motion_Timers[L_i](IN := VI_Motion_Sensors[L_i], PT := T#5m, VI_System_Time_MS := VI_System_Time_MS);

    // Сброс ручного переопределения, когда комната становится пустой (задний фронт таймера движения)
    IF L_Prev_Motion_Q[L_i] AND NOT L_Motion_Timers[L_i].Q THEN
        L_Manual_Override[L_i] := FALSE;
    END_IF;
    L_Prev_Motion_Q[L_i] := L_Motion_Timers[L_i].Q;

    IF L_Motion_Timers[L_i].Q THEN
        IF NOT L_Manual_Override[L_i] THEN
            L_Light_States[L_i] := TRUE;
        END_IF;
    ELSE
        // Выключаем свет только если нет ручного переопределения
        IF NOT L_Manual_Override[L_i] THEN
            L_Light_States[L_i] := FALSE;
        END_IF;
    END_IF;

    // Приоритет 3: Симуляция (только в режиме Away)
    IF L_Effective_Scenario = E_SCENARIO_TYPE.SCENARIO_AWAY AND L_Effective_Simulation_Active THEN
        L_Light_States[L_i] := VI_Simulation_Lights[L_i];
    END_IF;

    // Приоритет 4: Ручное управление и правила
    IF VI_Manual_Light_Override[L_i] > 0 THEN
        VO_Lighting_Levels[L_i] := VI_Manual_Light_Override[L_i];
    ELSIF L_Rule_Light_Active THEN
        VO_Lighting_Levels[L_i] := L_Rule_Light_Val;
    ELSE
        VO_Lighting_Levels[L_i] := SEL(L_Light_States[L_i], 0, L_Base_Light);
    END_IF;

    // 5. Мокрые зоны
    IF VI_Wet_Zone_Map[L_i] AND L_Wet_Zone_Idx <= GVL_CONSTANTS.C_MAX_WET_ZONES THEN
        VO_Wet_Zone_Light_Active[L_Wet_Zone_Idx] := (VO_Lighting_Levels[L_i] > 10);
        L_Wet_Zone_Idx := L_Wet_Zone_Idx + 1;
    END_IF;
END_FOR;

// 3. Управление шторами
FOR L_i := 1 TO GVL_CONSTANTS.C_MAX_BLINDS DO
    L_Rule_Blinds_Active := FALSE;
    L_Rule_Blinds_Val := 0;

    // Проверка правил
    FOR L_j := 1 TO GVL_CONSTANTS.C_MAX_RULES DO
        IF VI_Rule_Actions[L_j].Active AND VI_Rule_Actions[L_j].Target_ID = L_i THEN
            IF VI_Rule_Actions[L_j].Action_Type = E_Rule_Action_Type.ACTION_SET_BLINDS THEN
                L_Rule_Blinds_Active := TRUE;
                L_Rule_Blinds_Val := REAL_TO_BYTE(VI_Rule_Actions[L_j].Value);
            END_IF;
        END_IF;
    END_FOR;

    // Приоритет 1: Ручное управление
    IF VI_Manual_Blinds_Override[L_i] > 0 THEN
        VO_Blinds_Positions[L_i] := VI_Manual_Blinds_Override[L_i];
    // Приоритет 2: Правила
    ELSIF L_Rule_Blinds_Active THEN
        VO_Blinds_Positions[L_i] := L_Rule_Blinds_Val;
    // Приоритет 3: Сценарий
    ELSE
        VO_Blinds_Positions[L_i] := L_Base_Blinds;
    END_IF;
END_FOR;

// ========================================
// Lighting V2 shadow execution (phase2)
// ========================================
fbLightingV2Staging(
    VI_Zone_ID := 1,
    VI_Enable := (VO_Lighting_Levels[1] > 0),
    VI_Brightness_Setpoint := BYTE_TO_REAL(VO_Lighting_Levels[1]),
    VI_Scene_ID := TO_INT(L_Effective_Scenario),
    VI_Manual_Override := (VI_Manual_Light_Override[1] > 0),
    VI_Transition_Time_MS := 5000,

    VI_Is_Active := (VO_Lighting_Levels[1] > 0),
    VI_Brightness_Actual := BYTE_TO_REAL(VO_Lighting_Levels[1]),
    VI_Motion_Active := VI_Motion_Sensors[1],
    VI_Ambient_Lux := 0.0,
    VI_Alarm_Active := GVL_STATE.G_Lighting_IO_Fault OR GVL_STATE.G_Lighting_Subsystem_Degraded,

    VO_Command_Shadow => L_Lighting_V2_Command_Shadow,
    VO_State_Shadow => L_Lighting_V2_State_Shadow
);

// ========================================
// Lighting V2 shadow validation
// ========================================
IF ABS(BYTE_TO_REAL(VO_Lighting_Levels[1]) - L_Lighting_V2_Command_Shadow.Brightness_Setpoint) > 0.1 THEN
    L_Lighting_V2_Shadow_Diff_Found := TRUE;
END_IF;
IF ABS(BYTE_TO_REAL(VO_Lighting_Levels[1]) - L_Lighting_V2_State_Shadow.Brightness_Actual) > 0.1 THEN
    L_Lighting_V2_Shadow_Diff_Found := TRUE;
END_IF;
IF VI_Motion_Sensors[1] <> L_Lighting_V2_State_Shadow.Motion_Active THEN
    L_Lighting_V2_Shadow_Diff_Found := TRUE;
END_IF;

// Guarded Lighting V2 enable
IF L_Lighting_V2_Switch_Enabled THEN
    IF NOT L_Lighting_V2_Shadow_Diff_Found THEN
        L_Lighting_V2_Path_Ready := TRUE;
        L_Lighting_Using_Legacy_Fallback := FALSE;
    ELSE
        L_Lighting_V2_Path_Ready := FALSE;
        L_Lighting_Using_Legacy_Fallback := TRUE;
    END_IF;
ELSE
    L_Lighting_V2_Path_Ready := FALSE;
    L_Lighting_Using_Legacy_Fallback := TRUE;
END_IF;

// ========================================
// Blinds V2 shadow execution (phase2)
// ========================================
fbBlindsV2Staging(
    VI_Blind_ID := 1,
    VI_Enable := TRUE,
    VI_Position_Setpoint := VO_Blinds_Positions[1],
    VI_Manual_Override := (VI_Manual_Blinds_Override[1] > 0),
    VI_Scenario_ID := TO_INT(L_Effective_Scenario),
    VI_Safety_Mode := FALSE,

    VI_Position_Actual := VO_Blinds_Positions[1],
    VI_Manual_Override_Active := (VI_Manual_Blinds_Override[1] > 0),
    VI_Is_Moving := FALSE,
    VI_Alarm_Active := GVL_STATE.G_Lighting_IO_Fault,

    VO_Command_Shadow => L_Blinds_V2_Command_Shadow,
    VO_State_Shadow => L_Blinds_V2_State_Shadow
);

// Blinds validation
IF VO_Blinds_Positions[1] <> L_Blinds_V2_Command_Shadow.Position_Setpoint THEN
    L_Blinds_V2_Shadow_Diff_Found := TRUE;
END_IF;
IF VO_Blinds_Positions[1] <> L_Blinds_V2_State_Shadow.Position_Actual THEN
    L_Blinds_V2_Shadow_Diff_Found := TRUE;
END_IF;

// Guarded Blinds V2 enable
IF L_Blinds_V2_Switch_Enabled THEN
    IF NOT L_Blinds_V2_Shadow_Diff_Found THEN
        L_Blinds_V2_Path_Ready := TRUE;
        L_Blinds_Using_Legacy_Fallback := FALSE;
    ELSE
        L_Blinds_V2_Path_Ready := FALSE;
        L_Blinds_Using_Legacy_Fallback := TRUE;
    END_IF;
ELSE
    L_Blinds_V2_Path_Ready := FALSE;
    L_Blinds_Using_Legacy_Fallback := TRUE;
END_IF;

END_FUNCTION_BLOCK
// >>> BULK_SYNC_ANCHOR: FB_Lighting_Blinds_Manager <<<

(* ---- FB_PLC_Heartbeat.st ---- *)
FUNCTION_BLOCK FB_PLC_Heartbeat
VAR_INPUT
    VI_Local_ID : BYTE; // Идентификатор данного ПЛК (1 - ПЛК А, 2 - ПЛК B)
    VI_System_Time : UDINT; // Текущее системное время (мс)
    VI_Remote_Pulse : BOOL; // Сигнал пульса от партнерского ПЛК
    VI_Remote_Is_Active : BOOL; // Статус активности партнерского ПЛК (ТЗ 8.3)
    VI_Gateway_Ping_OK : BOOL; // Флаг доступности сетевого шлюза (ТЗ 8.3)
END_VAR
VAR_OUTPUT
    VO_Is_Active : BOOL; // Выход: Данный ПЛК является ведущим (Active)
    VO_RTT_MS : UDINT; // Текущая задержка связи между ПЛК (Round Trip Time)
    VO_Loss_Count : UDINT; // Счетчик потерь пакетов связи (ТЗ 8.4)
    VO_Max_RTT : UDINT; // Максимальная зафиксированная задержка связи
END_VAR
VAR
    L_Last_Pulse : BOOL; // Предыдущее состояние сигнала пульса
    L_Last_Pulse_Time : UDINT; // Время последнего изменения сигнала пульса
    L_Timeout : UDINT := 500; // Порог таймаута связи (500 мс по ТЗ 8.1)
    L_Pulse_Send_Time : UDINT; // Время отправки собственного пульса
    L_Last_Loss_Time : UDINT; // Время последней фиксации потери связи
    L_Elapsed_Time : UDINT;
END_VAR

// Вспомогательная функция для безопасного вычисления разницы времени
L_Elapsed_Time := (VI_System_Time - L_Last_Pulse_Time);

// 1. Мониторинг "сердцебиения" и расчет сетевых задержек (ТЗ 8.4)
IF VI_Remote_Pulse <> L_Last_Pulse THEN
    // Вычисляем время между изменениями сигнала
    VO_RTT_MS := L_Elapsed_Time;
    // Фиксируем пиковые задержки для диагностики сети
    IF VO_RTT_MS > VO_Max_RTT THEN VO_Max_RTT := VO_RTT_MS; END_IF;
    L_Last_Pulse := VI_Remote_Pulse;
    L_Last_Pulse_Time := VI_System_Time;
    L_Elapsed_Time := 0; // Сбрасываем после обновления
END_IF;

// Подсчет статистики потерь связи (ТЗ 8.4)
IF L_Elapsed_Time > L_Timeout THEN
    IF (VI_System_Time - L_Last_Loss_Time) >= 1000 THEN
        VO_Loss_Count := VO_Loss_Count + 1;
        L_Last_Loss_Time := VI_System_Time;
    END_IF;
ELSE
    L_Last_Loss_Time := VI_System_Time;
END_IF;

// 2. Логика определения роли (Active/Standby) и предотвращение Split-Brain (ТЗ 8.3)
// Уровень 1: Проверка наличия связи с партнером
IF L_Elapsed_Time < L_Timeout THEN
    // Связь есть: Договариваемся о ролях на основе приоритета ID
    IF VI_Local_ID = 1 THEN
        VO_Is_Active := TRUE; // ПЛК А всегда активен при наличии связи
    ELSE
        VO_Is_Active := NOT VI_Remote_Is_Active; // ПЛК B активен только если А не активен
    END_IF;
ELSE
    // Связи нет: Пытаемся определить, кто из нас "живее"
    // Уровень 3: Если связи с партнером нет, проверяем доступность внешнего шлюза
    IF VI_Local_ID = 1 THEN
        // ПЛК А становится активным всегда при потере связи с партнером (fallback)
        VO_Is_Active := TRUE;
    ELSE
        // ПЛК B ждет таймаут удержания роли (2 секунды), прежде чем стать активным
        IF L_Elapsed_Time >= 2000 THEN
            // ПЛК B берет управление если он видит шлюз, а связи с А нет.
            // Если шлюз недоступен, B ждет дольше (fallback).
            IF VI_Gateway_Ping_OK THEN
                VO_Is_Active := TRUE;
            ELSIF L_Elapsed_Time >= 5000 THEN
                VO_Is_Active := TRUE; // Fallback: ПЛК А мертв и шлюз мертв
            ELSE
                VO_Is_Active := FALSE;
            END_IF;
        ELSE
            VO_Is_Active := FALSE;
        END_IF;
    END_IF;
END_IF;

(* ---- FB_Presence_Simulator.st ---- *)
FUNCTION_BLOCK FB_Presence_Simulator
VAR_INPUT
    VI_Enabled : BOOL;
    VI_Intensity : REAL;
    VI_System_Time : UDINT;
    VI_Use_Playback : BOOL; // Новый режим воспроизведения
END_VAR
VAR_OUTPUT
    VO_Light_States : ARRAY[1..32] OF BOOL;
END_VAR
VAR
    fbPlayback : FB_Presence_Playback;
END_VAR

IF VI_Enabled THEN
    IF VI_Use_Playback THEN
        fbPlayback(VI_Mode_Record := FALSE, VI_Time_Index := VI_System_Time MOD 604800000, VO_Light_Outputs => VO_Light_States);
    ELSE
        // Старая логика случайной симуляции
        VO_Light_States[1] := (VI_System_Time MOD 100000 > 50000);
    END_IF;
END_IF;

(* ---- FB_Security_Alarm.st ---- *)
FUNCTION_BLOCK FB_Security_Alarm
VAR_INPUT
    VI_Armed       : BOOL;
    VI_Motion      : BOOL;
    VI_Door        : BOOL;
    VI_Delay_MS    : UDINT := 30000;
    VI_System_Time : UDINT;
END_VAR
VAR_OUTPUT
    VO_Alarm       : BOOL;
END_VAR
VAR
    L_Trigger_Time : UDINT;
    L_Triggered    : BOOL;
END_VAR

IF VI_Armed AND (VI_Motion OR VI_Door) AND NOT L_Triggered THEN
    L_Triggered := TRUE;
    L_Trigger_Time := VI_System_Time;
END_IF;

IF L_Triggered AND ((SEL(VI_System_Time >= L_Trigger_Time, VI_System_Time - L_Trigger_Time, (4294967295 - L_Trigger_Time) + VI_System_Time + 1)) >= VI_Delay_MS) THEN
    VO_Alarm := TRUE;
ELSIF NOT VI_Armed THEN
    L_Triggered := FALSE;
    VO_Alarm := FALSE;
END_IF;

(* ---- FB_Security_System_Manager.st ---- *)
FUNCTION_BLOCK FB_Security_System_Manager
VAR_INPUT
    VI_System_Time_MS : UDINT; // Системное время (мс)
    VI_IsActivePLC : BOOL; // Флаг: Данный ПЛК является ведущим
    VI_Arm_Request : BOOL; // Запрос на постановку под охрану
    VI_Disarm_Request : BOOL; // Запрос на снятие с охраны
    VI_PIN_Code : STRING(4); // ПИН-код для авторизации
    VI_RFID_Tag : STRING(20); // RFID/NFC метка для авторизации
    VI_2FA_Code : STRING(6); // Код двухфакторной аутентификации
    VI_Config : ST_Security_Global_Config; // Конфигурация охранной системы
    VI_Current_TOD : TOD; // Текущее время суток (от FB_Astro_Timer)
END_VAR
VAR_IN_OUT
    VI_Motion_Sensors : ARRAY[1..16] OF BOOL; // Датчики движения
    VI_Door_Sensors : ARRAY[1..GVL_CONSTANTS.C_MAX_DOOR_SENSORS] OF BOOL; // Датчики открытия дверей (герконы)
    VI_Window_Sensors : ARRAY[1..16] OF BOOL; // Датчики открытия окон (герконы)
    VI_Bypass_Motion : ARRAY[1..16] OF BOOL; // Байпас датчиков движения
    VI_Bypass_Doors : ARRAY[1..GVL_CONSTANTS.C_MAX_DOOR_SENSORS] OF BOOL; // Байпас дверей
    VI_Bypass_Windows : ARRAY[1..16] OF BOOL; // Байпас окон
END_VAR
VAR_OUTPUT
    VO_Armed : BOOL; // Статус: Система под охраной
    VO_Alarm_Active : BOOL; // Статус: Тревога активна
    VO_Siren_Active : BOOL; // Команда: Включить сирену
    VO_Status_Msg : STRING(200); // Строковое сообщение о статусе
    VO_Send_Code_Req : BOOL; // Запрос на отправку кода 2FA
    VO_Code_To_Send : STRING(6); // Сгенерированный код 2FA для отправки
END_VAR
VAR
    L_i : INT;
    L_Any_Sensor_Active : BOOL;
    L_Arm_Delay_Timer : FB_System_Timer;
    L_Alarm_Delay_Timer : FB_System_Timer;
    L_Arming_In_Progress : BOOL;
    L_Valid_PIN : BOOL;
    fbAccessCode : FB_AccessCode_Manager;
    fbTwoFactor : FB_TwoFactor_Auth;
    L_2FA_Required : BOOL;
    L_Disarm_Pending : BOOL;
    L_Reset_2FA : BOOL;
    L_Auto_Arm_Trigger : BOOL;
    R_Trig_Auto_Arm : R_TRIG;
END_VAR

IF NOT VI_IsActivePLC THEN RETURN; END_IF;

// 1. Проверка PIN-кода или RFID-метки через менеджер кодов
fbAccessCode(
    VI_System_Time_MS := VI_System_Time_MS,
    VI_IsActivePLC := VI_IsActivePLC,
    VI_Code_To_Check := VI_PIN_Code,
    VI_RFID_To_Check := VI_RFID_Tag,
    VI_Access_Codes := GVL_RETAIN.G_Access_Codes,
    VI_RFID_Tags := GVL_RETAIN.G_RFID_Tags,
    VO_Code_Valid => L_Valid_PIN
);

// 2. Логика постановки на охрану (с задержкой на выход)
L_Auto_Arm_Trigger := FALSE;
IF VI_Config.auto_arm_enabled THEN
    IF VI_Current_TOD >= UDINT_TO_TOD(VI_Config.auto_arm_time_ms) THEN
        L_Auto_Arm_Trigger := TRUE;
    END_IF;
END_IF;
R_Trig_Auto_Arm(CLK := L_Auto_Arm_Trigger);

IF ((VI_Arm_Request AND L_Valid_PIN) OR R_Trig_Auto_Arm.Q) AND NOT VO_Armed AND NOT L_Arming_In_Progress THEN
    // Проверка, что все двери/окна закрыты перед постановкой (с учетом байпаса)
    L_Any_Sensor_Active := FALSE;
    FOR L_i := 1 TO GVL_CONSTANTS.C_MAX_DOOR_SENSORS DO IF VI_Door_Sensors[L_i] AND NOT VI_Bypass_Doors[L_i] THEN L_Any_Sensor_Active := TRUE; END_IF; END_FOR;
    FOR L_i := 1 TO GVL_CONSTANTS.C_MAX_CLIMATE_ZONES DO IF VI_Window_Sensors[L_i] AND NOT VI_Bypass_Windows[L_i] THEN L_Any_Sensor_Active := TRUE; END_IF; END_FOR;

    IF NOT L_Any_Sensor_Active THEN
        L_Arming_In_Progress := TRUE;
        VO_Status_Msg := 'Постановка на охрану. Покиньте помещение.';
    ELSE
        VO_Status_Msg := 'Ошибка постановки: Открыты двери или окна';
    END_IF;
END_IF;

L_Arm_Delay_Timer(IN := L_Arming_In_Progress, PT := TO_TIME(VI_Config.exit_delay_seconds * 1000), VI_System_Time_MS := VI_System_Time_MS);
IF L_Arm_Delay_Timer.Q THEN
    L_Arming_In_Progress := FALSE;
    VO_Armed := TRUE;
    VO_Status_Msg := 'Система под охраной';
END_IF;

// 3. Логика снятия с охраны с 2FA
IF VI_Disarm_Request AND L_Valid_PIN AND VO_Armed THEN
    IF VI_Config.enable_2fa THEN
        L_Disarm_Pending := TRUE;
        L_2FA_Required := TRUE;
        VO_Status_Msg := 'Ожидание 2FA для снятия с охраны';
    ELSE
        // Снятие без 2FA
        VO_Armed := FALSE;
        VO_Alarm_Active := FALSE;
        VO_Siren_Active := FALSE;
        L_Arming_In_Progress := FALSE;
        VO_Status_Msg := 'Система снята с охраны';
    END_IF;
END_IF;

fbTwoFactor(
    VI_System_Time_MS := VI_System_Time_MS,
    VI_Start_Auth := L_2FA_Required,
    VI_Method := E_TwoFactor_Method.TF_METHOD_TOTP, // Для примера
    VI_User_Code := VI_2FA_Code, // Используем отдельный вход для 2FA кода
    VI_Reset_Success := L_Reset_2FA
);

VO_Send_Code_Req := fbTwoFactor.VO_Send_Code_Req;
VO_Code_To_Send := fbTwoFactor.VO_Code_To_Send;

IF L_Disarm_Pending AND fbTwoFactor.VO_State.Is_Success THEN
    VO_Armed := FALSE;
    VO_Alarm_Active := FALSE;
    VO_Siren_Active := FALSE;
    L_Arming_In_Progress := FALSE;
    L_Disarm_Pending := FALSE;
    L_2FA_Required := FALSE;
    L_Reset_2FA := TRUE;
    VO_Status_Msg := 'Система снята с охраны';
ELSIF L_Disarm_Pending AND fbTwoFactor.VO_State.Is_Locked THEN
    L_Disarm_Pending := FALSE;
    L_2FA_Required := FALSE;
    L_Reset_2FA := FALSE;
    VO_Status_Msg := 'Ошибка 2FA: Превышено количество попыток';
ELSE
    L_Reset_2FA := FALSE;
END_IF;

// 4. Логика тревоги (с задержкой на вход)
IF VO_Armed THEN
    L_Any_Sensor_Active := FALSE;
    FOR L_i := 1 TO GVL_CONSTANTS.C_MAX_CLIMATE_ZONES DO IF VI_Motion_Sensors[L_i] AND NOT VI_Bypass_Motion[L_i] THEN L_Any_Sensor_Active := TRUE; END_IF; END_FOR;
    FOR L_i := 1 TO GVL_CONSTANTS.C_MAX_DOOR_SENSORS DO IF VI_Door_Sensors[L_i] AND NOT VI_Bypass_Doors[L_i] THEN L_Any_Sensor_Active := TRUE; END_IF; END_FOR;
    FOR L_i := 1 TO GVL_CONSTANTS.C_MAX_CLIMATE_ZONES DO IF VI_Window_Sensors[L_i] AND NOT VI_Bypass_Windows[L_i] THEN L_Any_Sensor_Active := TRUE; END_IF; END_FOR;

    // Защелкиваем факт нарушения периметра, чтобы кратковременное срабатывание датчика не сбрасывало таймер
    IF L_Any_Sensor_Active THEN
        L_Alarm_Delay_Timer.IN := TRUE;
    END_IF;

    L_Alarm_Delay_Timer(PT := TO_TIME(VI_Config.entry_delay_seconds * 1000), VI_System_Time_MS := VI_System_Time_MS);

    IF L_Alarm_Delay_Timer.Q THEN
        VO_Alarm_Active := TRUE;
        VO_Siren_Active := TRUE;
        VO_Status_Msg := 'ТРЕВОГА! Нарушение периметра';
    ELSIF L_Alarm_Delay_Timer.IN THEN
        VO_Status_Msg := 'Внимание! Введите PIN-код для отмены тревоги';
    END_IF;
ELSE
    L_Alarm_Delay_Timer(IN := FALSE, PT := T#0s, VI_System_Time_MS := VI_System_Time_MS); // Сброс таймера при снятии с охраны
END_IF;
// >>> BULK_SYNC_ANCHOR: FB_Security_System_Manager <<<

(* ---- FB_Sensor_Analog_Processing.st ---- *)
FUNCTION_BLOCK FB_Sensor_Analog_Processing
VAR_INPUT
    VI_Raw_Value : WORD; // Raw value from module (e.g., 0-27648)
    VI_Sensor_Type : INT := 0; // 0: 4-20mA, 1: 0-10V, 2: PT100/1000 (direct temp * 10)
    VI_Min_Scale : REAL; // Minimum scale value (e.g., 0 bar)
    VI_Max_Scale : REAL; // Maximum scale value (e.g., 10 bar)
    VI_Offset : REAL; // Calibration offset
    VI_Multiplier : REAL := 1.0; // Calibration multiplier
    VI_Filter_Time_MS : UDINT := GVL_CONSTANTS.C_MS_IN_SECOND; // Filtering time
    VI_System_Time_MS : UDINT; // System time in ms
    VI_Fallback_Mode : INT := 0; // 0: Hold last good value, 1: Use default value
    VI_Default_Value : REAL := 0.0; // Default value for fallback mode 1
END_VAR
VAR_OUTPUT
    VO_Value : REAL; // Processed value
    VO_Error : BOOL; // Sensor error (open/short circuit)
    VO_Diag_Code : WORD; // Diagnostic code (0: OK, 1: Open circuit, 2: Short circuit, 3: Out of range)
END_VAR
VAR
    L_Scaled : REAL;
    L_Filtered : REAL;
    L_History : ARRAY[0..9] OF REAL; // Массив для скользящего среднего (10 значений)
    L_History_Idx : INT := 0;
    L_History_Sum : REAL := 0.0;
    L_History_Count : INT := 0;
    L_Last_Time : UDINT;
    L_DT : UDINT;
    L_First_Scan : BOOL := TRUE;
    L_i : INT;
END_VAR

// 1. Error checking and scaling based on sensor type
VO_Error := FALSE;
VO_Diag_Code := 0;

CASE VI_Sensor_Type OF
    0: // 4-20mA (NAMUR NE43: < 3.6mA or > 21mA)
        IF VI_Raw_Value < GVL_CONSTANTS.C_ANALOG_3_6MA_RAW THEN // < 3.6mA (Open circuit)
            VO_Error := TRUE;
            VO_Diag_Code := 1;
        ELSIF VI_Raw_Value > GVL_CONSTANTS.C_ANALOG_21MA_RAW THEN // > 21mA (Short circuit)
            VO_Error := TRUE;
            VO_Diag_Code := 2;
        ELSE
            // 4mA = 5529, 20mA = 27648
            L_Scaled := VI_Min_Scale + (TO_REAL(VI_Raw_Value - GVL_CONSTANTS.C_ANALOG_4MA_RAW) / TO_REAL(GVL_CONSTANTS.C_ANALOG_RAW_MAX - GVL_CONSTANTS.C_ANALOG_4MA_RAW)) * (VI_Max_Scale - VI_Min_Scale);
        END_IF;

    1: // 0-10V (0-27648)
        IF VI_Raw_Value > GVL_CONSTANTS.C_ANALOG_10V_MAX_RAW THEN // Out of range
            VO_Error := TRUE;
            VO_Diag_Code := 3;
        ELSE
            L_Scaled := VI_Min_Scale + (TO_REAL(VI_Raw_Value) / TO_REAL(GVL_CONSTANTS.C_ANALOG_RAW_MAX)) * (VI_Max_Scale - VI_Min_Scale);
        END_IF;

    2: // PT100/1000 (Direct temperature * 10, e.g., 255 = 25.5C)
        // Typically, 16-bit signed integer for temperature
        IF VI_Raw_Value = 16#7FFF OR VI_Raw_Value = 16#8000 THEN // Sensor error codes
            VO_Error := TRUE;
            VO_Diag_Code := 1;
        ELSE
            L_Scaled := TO_REAL(TO_INT(VI_Raw_Value)) / 10.0;
            IF L_Scaled < VI_Min_Scale OR L_Scaled > VI_Max_Scale THEN
                VO_Error := TRUE;
                VO_Diag_Code := 3;
            END_IF;
        END_IF;

    ELSE
        VO_Error := TRUE;
        VO_Diag_Code := 16#FFFF; // Unknown sensor type
END_CASE;

// 2. Fallback handling
IF VO_Error THEN
    IF VI_Fallback_Mode = 1 THEN
        VO_Value := VI_Default_Value;
    END_IF;
    // If VI_Fallback_Mode = 0, VO_Value retains its last good value (L_Filtered)
    RETURN;
END_IF;

// 3. Calibration
L_Scaled := (L_Scaled * VI_Multiplier) + VI_Offset;

// 4. Moving Average Filter (ТЗ 1.2)
IF L_First_Scan THEN
    L_Filtered := L_Scaled;
    L_First_Scan := FALSE;
    L_Last_Time := VI_System_Time_MS;

    // Инициализация массива истории
    FOR L_i := 0 TO 9 DO
        L_History[L_i] := L_Scaled;
    END_FOR;
    L_History_Sum := L_Scaled * 10.0;
    L_History_Count := 10;
    L_History_Idx := 0;
END_IF;

L_DT := (SEL(VI_System_Time_MS >= L_Last_Time, VI_System_Time_MS - L_Last_Time, (4294967295 - L_Last_Time) + VI_System_Time_MS + 1));
IF VI_Filter_Time_MS = 0 THEN
    L_Filtered := L_Scaled;
    L_Last_Time := VI_System_Time_MS;
ELSIF L_DT >= (VI_Filter_Time_MS / 10) THEN // Обновляем 10 раз за время фильтрации
    // Вычитаем старое значение
    L_History_Sum := L_History_Sum - L_History[L_History_Idx];

    // Добавляем новое значение
    L_History[L_History_Idx] := L_Scaled;
    L_History_Sum := L_History_Sum + L_Scaled;

    // Сдвигаем индекс
    L_History_Idx := (L_History_Idx + 1) MOD 10;

    // Вычисляем среднее
    L_Filtered := L_History_Sum / 10.0;

    L_Last_Time := VI_System_Time_MS;
END_IF;

VO_Value := L_Filtered;

(* ---- FB_Sensor_Distribution.st ---- *)
FUNCTION_BLOCK FB_Sensor_Distribution
VAR_INPUT
    VI_Raw_Temp : REAL;
    VI_Raw_Hum  : REAL;
    VI_Raw_CO2  : REAL;
END_VAR
VAR_OUTPUT
    VO_Temp_Heating : REAL;
    VO_Temp_Vent    : REAL;
    VO_Hum_Vent     : REAL;
    VO_CO2_Vent     : REAL;
END_VAR

// Распределение данных по подсистемам
VO_Temp_Heating := VI_Raw_Temp;
VO_Temp_Vent    := VI_Raw_Temp;
VO_Hum_Vent     := VI_Raw_Hum;
VO_CO2_Vent     := VI_Raw_CO2;

(* ---- FB_State_Snapshot_Manager.st ---- *)
FUNCTION_BLOCK FB_State_Snapshot_Manager
VAR_INPUT
    VI_System_Time_MS : UDINT;
    VI_Trigger_Event  : BOOL; // Сигнал на создание снимка
    VI_Event_Code     : WORD;
    VI_Current_State  : ST_State_Snapshot;
END_VAR
VAR_OUTPUT
    VO_Snapshot_Saved : BOOL;
END_VAR
VAR
    L_Snapshot_Buffer : ARRAY[1..GVL_CONSTANTS.C_MAX_STATE_SNAPSHOTS] OF ST_State_Snapshot;
    L_Write_Idx       : INT := 1;
END_VAR

IF VI_Trigger_Event THEN
    L_Snapshot_Buffer[L_Write_Idx] := VI_Current_State;
    L_Snapshot_Buffer[L_Write_Idx].timestamp_ms := VI_System_Time_MS;
    L_Snapshot_Buffer[L_Write_Idx].trigger_event_code := VI_Event_Code;

    L_Write_Idx := (L_Write_Idx MOD GVL_CONSTANTS.C_MAX_STATE_SNAPSHOTS) + 1;
    VO_Snapshot_Saved := TRUE;
ELSE
    VO_Snapshot_Saved := FALSE;
END_IF;

(* ---- FB_System_Health.st ---- *)
FUNCTION_BLOCK FB_System_Health
VAR_INPUT
    VI_Smoke_Detected      : BOOL;
    VI_Gas_Detected        : BOOL;
    VI_CO_Warning_Level    : BOOL;
    VI_CO_Alarm_Level      : BOOL;
    VI_Leak_Detected       : BOOL;

    VI_Sensor_Fault        : BOOL := FALSE;
    VI_IO_Offline          : BOOL := FALSE;
    VI_Comm_Fault          : BOOL := FALSE;
    VI_Watchdog_Fault      : BOOL := FALSE;
    VI_Subsystem_Fault     : BOOL := FALSE;
END_VAR

VAR_OUTPUT
    VO_System_Severity     : E_System_Severity;
    VO_Root_Cause          : E_System_Root_Cause;

    // compatibility outputs for existing orchestration
    VO_Sensor_Fault        : BOOL;
    VO_IO_Fault            : BOOL;
    VO_Comm_Fault          : BOOL;
    VO_Subsystem_Degraded  : BOOL;

    VO_First_Fault_Active  : BOOL;
    VO_First_Fault_Type    : INT;
    VO_First_Fault_Source  : INT;
END_VAR

VO_Sensor_Fault := VI_Sensor_Fault;
VO_IO_Fault := VI_IO_Offline;
VO_Comm_Fault := VI_Comm_Fault;
VO_Subsystem_Degraded := VI_Subsystem_Fault;

VO_System_Severity := E_System_Severity.SEV_NORMAL;
VO_Root_Cause := E_System_Root_Cause.ROOT_NONE;
VO_First_Fault_Active := FALSE;
VO_First_Fault_Type := 0;
VO_First_Fault_Source := 0;

// Priority: FIRE > GAS > CO > WATER > diagnostics
IF VI_Smoke_Detected THEN
    VO_System_Severity := E_System_Severity.SEV_CRITICAL;
    VO_Root_Cause := E_System_Root_Cause.ROOT_FIRE;
    VO_First_Fault_Active := TRUE;
    VO_First_Fault_Type := 5;

ELSIF VI_Gas_Detected THEN
    VO_System_Severity := E_System_Severity.SEV_CRITICAL;
    VO_Root_Cause := E_System_Root_Cause.ROOT_GAS_LEAK;
    VO_First_Fault_Active := TRUE;
    VO_First_Fault_Type := 6;

ELSIF VI_CO_Alarm_Level THEN
    VO_System_Severity := E_System_Severity.SEV_CRITICAL;
    VO_Root_Cause := E_System_Root_Cause.ROOT_CO_CRITICAL;
    VO_First_Fault_Active := TRUE;
    VO_First_Fault_Type := 7;

ELSIF VI_CO_Warning_Level THEN
    VO_System_Severity := E_System_Severity.SEV_WARNING;
    VO_Root_Cause := E_System_Root_Cause.ROOT_CO_WARNING;
    VO_First_Fault_Active := TRUE;
    VO_First_Fault_Type := 7;

ELSIF VI_Leak_Detected THEN
    VO_System_Severity := E_System_Severity.SEV_WARNING;
    VO_Root_Cause := E_System_Root_Cause.ROOT_WATER_LEAK;
    VO_First_Fault_Active := TRUE;
    VO_First_Fault_Type := 8;

ELSIF VI_Watchdog_Fault THEN
    VO_System_Severity := E_System_Severity.SEV_CRITICAL;
    VO_Root_Cause := E_System_Root_Cause.ROOT_WATCHDOG_FAULT;
    VO_First_Fault_Active := TRUE;
    VO_First_Fault_Type := 9;

ELSIF VI_IO_Offline THEN
    VO_System_Severity := E_System_Severity.SEV_DEGRADED;
    VO_Root_Cause := E_System_Root_Cause.ROOT_IO_OFFLINE;
    VO_First_Fault_Active := TRUE;
    VO_First_Fault_Type := 1;

ELSIF VI_Comm_Fault THEN
    VO_System_Severity := E_System_Severity.SEV_DEGRADED;
    VO_Root_Cause := E_System_Root_Cause.ROOT_COMM_FAULT;
    VO_First_Fault_Active := TRUE;
    VO_First_Fault_Type := 3;

ELSIF VI_Sensor_Fault THEN
    VO_System_Severity := E_System_Severity.SEV_DEGRADED;
    VO_Root_Cause := E_System_Root_Cause.ROOT_SENSOR_FAULT;
    VO_First_Fault_Active := TRUE;
    VO_First_Fault_Type := 2;

ELSIF VI_Subsystem_Fault THEN
    VO_System_Severity := E_System_Severity.SEV_DEGRADED;
    VO_Root_Cause := E_System_Root_Cause.ROOT_SUBSYSTEM_FAULT;
    VO_First_Fault_Active := TRUE;
    VO_First_Fault_Type := 4;
END_IF;
// >>> BULK_SYNC_ANCHOR: FB_System_Health <<<

(* ---- FB_TwoFactor_Auth.st ---- *)
FUNCTION_BLOCK FB_TwoFactor_Auth
VAR_INPUT
    VI_System_Time_MS : UDINT;
    VI_Start_Auth     : BOOL;
    VI_Method         : E_TwoFactor_Method;
    VI_User_Code      : STRING(6);
    VI_Reset_Success  : BOOL; // Сброс успешного состояния
END_VAR
VAR_OUTPUT
    VO_State          : ST_TwoFactor_Auth_State;
    VO_Send_Code_Req  : BOOL; // Запрос на отправку кода (например, через шлюз)
    VO_Code_To_Send   : STRING(6); // Сгенерированный код для отправки
END_VAR
VAR
    L_Generated_Code  : STRING(6) := '';
    L_Start_Time      : UDINT;
    R_Trig_Start      : R_TRIG;
    L_Prev_User_Code  : STRING(6);
    L_Lockout_Start_Time : UDINT; // Время начала блокировки
    fbHMAC            : FB_HMAC_SHA1;
    L_Elapsed_Time    : UDINT;
    L_Time_Step       : UDINT;
    L_Message         : ARRAY[0..7] OF BYTE;
    L_Key             : ARRAY[0..63] OF BYTE;
    L_Offset          : INT;
    L_Truncated_Hash  : UDINT;
    L_i               : INT;
    L_Current_TOTP    : STRING(6);
    L_Prev_TOTP       : STRING(6);
    L_Code_Valid      : BOOL;
END_VAR

R_Trig_Start(CLK := VI_Start_Auth);

IF VI_Reset_Success THEN
    VO_State.Is_Success := FALSE;
END_IF;

IF R_Trig_Start.Q AND NOT VO_State.is_pending AND NOT VO_State.Is_Locked THEN
    VO_State.is_pending := TRUE;
    VO_State.Auth_Method := VI_Method;
    L_Start_Time := VI_System_Time_MS;
    VO_State.Attempts_Left := 3;
    VO_State.Is_Success := FALSE;
    VO_State.Is_Locked := FALSE;
    L_Prev_User_Code := '';

    IF VI_Method <> E_TwoFactor_Method.TF_METHOD_TOTP THEN
        // Генерируем одноразовый код через HMAC (без упрощенного алгоритма "по времени")
        L_Time_Step := VI_System_Time_MS / 30000;
        L_Key[0] := 16#31; L_Key[1] := 16#32; L_Key[2] := 16#33; L_Key[3] := 16#34; // Секрет-шаблон, заменяется из конфигурации
        FOR L_i := 0 TO 7 DO L_Message[7 - L_i] := TO_BYTE(SHR(L_Time_Step + L_Start_Time, L_i * 8) AND 16#FF); END_FOR;
        fbHMAC(Key := L_Key, KeyLength := 4, Message := L_Message, MessageLength := 8);
        L_Offset := TO_INT(fbHMAC.Hash[19] AND 16#0F);
        L_Truncated_Hash := (SHL(TO_UDINT(fbHMAC.Hash[L_Offset] AND 16#7F), 24) OR SHL(TO_UDINT(fbHMAC.Hash[L_Offset+1] AND 16#FF), 16) OR SHL(TO_UDINT(fbHMAC.Hash[L_Offset+2] AND 16#FF), 8) OR TO_UDINT(fbHMAC.Hash[L_Offset+3] AND 16#FF));
        L_Generated_Code := UDINT_TO_STRING(L_Truncated_Hash MOD 1000000);
        WHILE LEN(L_Generated_Code) < 6 DO
            L_Generated_Code := CONCAT('0', L_Generated_Code);
        END_WHILE;

        VO_Code_To_Send := L_Generated_Code;
        VO_Send_Code_Req := TRUE;
    ELSE
        // Для TOTP код не отправляем
        VO_Code_To_Send := '';
        VO_Send_Code_Req := FALSE;
    END_IF;
ELSE
    VO_Send_Code_Req := FALSE;
END_IF;

IF VO_State.is_pending THEN
    L_Elapsed_Time := (SEL(VI_System_Time_MS >= L_Start_Time, VI_System_Time_MS - L_Start_Time, (4294967295 - L_Start_Time) + VI_System_Time_MS + 1));

    IF L_Elapsed_Time < (GVL_CONSTANTS.C_MS_IN_MINUTE * 5) THEN
        VO_State.Time_Left_S := TO_UINT(((GVL_CONSTANTS.C_MS_IN_MINUTE * 5) - L_Elapsed_Time) / 1000);
    ELSE
        VO_State.Time_Left_S := 0;
    END_IF;

    IF VI_User_Code <> '' AND VI_User_Code <> L_Prev_User_Code THEN
        L_Code_Valid := FALSE;

        IF VI_Method = E_TwoFactor_Method.TF_METHOD_TOTP THEN
            // Вычисляем TOTP для текущего шага времени (30 секунд)
            L_Time_Step := VI_System_Time_MS / 30000;

            // Подготовка ключа (в реальном проекте берется из GVL_CONFIG)
            L_Key[0] := 16#31; L_Key[1] := 16#32; L_Key[2] := 16#33; L_Key[3] := 16#34; // '1234'

            // Проверка текущего шага
            FOR L_i := 0 TO 7 DO L_Message[7 - L_i] := TO_BYTE(SHR(L_Time_Step, L_i * 8) AND 16#FF); END_FOR;
            fbHMAC(Key := L_Key, KeyLength := 4, Message := L_Message, MessageLength := 8);
            L_Offset := TO_INT(fbHMAC.Hash[19] AND 16#0F);
            L_Truncated_Hash := (SHL(TO_UDINT(fbHMAC.Hash[L_Offset] AND 16#7F), 24) OR SHL(TO_UDINT(fbHMAC.Hash[L_Offset+1] AND 16#FF), 16) OR SHL(TO_UDINT(fbHMAC.Hash[L_Offset+2] AND 16#FF), 8) OR TO_UDINT(fbHMAC.Hash[L_Offset+3] AND 16#FF));
            L_Current_TOTP := UDINT_TO_STRING(L_Truncated_Hash MOD 1000000);
            WHILE LEN(L_Current_TOTP) < 6 DO L_Current_TOTP := CONCAT('0', L_Current_TOTP); END_WHILE;

            // Проверка предыдущего шага (для компенсации рассинхронизации)
            FOR L_i := 0 TO 7 DO L_Message[7 - L_i] := TO_BYTE(SHR(L_Time_Step - 1, L_i * 8) AND 16#FF); END_FOR;
            fbHMAC(Key := L_Key, KeyLength := 4, Message := L_Message, MessageLength := 8);
            L_Offset := TO_INT(fbHMAC.Hash[19] AND 16#0F);
            L_Truncated_Hash := (SHL(TO_UDINT(fbHMAC.Hash[L_Offset] AND 16#7F), 24) OR SHL(TO_UDINT(fbHMAC.Hash[L_Offset+1] AND 16#FF), 16) OR SHL(TO_UDINT(fbHMAC.Hash[L_Offset+2] AND 16#FF), 8) OR TO_UDINT(fbHMAC.Hash[L_Offset+3] AND 16#FF));
            L_Prev_TOTP := UDINT_TO_STRING(L_Truncated_Hash MOD 1000000);
            WHILE LEN(L_Prev_TOTP) < 6 DO L_Prev_TOTP := CONCAT('0', L_Prev_TOTP); END_WHILE;

            IF VI_User_Code = L_Current_TOTP OR VI_User_Code = L_Prev_TOTP THEN
                L_Code_Valid := TRUE;
            END_IF;
        ELSE
            IF VI_User_Code = L_Generated_Code THEN
                L_Code_Valid := TRUE;
            END_IF;
        END_IF;

        IF L_Code_Valid THEN
            VO_State.Is_Success := TRUE;
            VO_State.is_pending := FALSE;
        ELSE
            IF VO_State.Attempts_Left > 0 THEN
                VO_State.Attempts_Left := VO_State.Attempts_Left - 1;
            END_IF;

            IF VO_State.Attempts_Left = 0 THEN
                VO_State.Is_Locked := TRUE;
                VO_State.is_pending := FALSE;
                L_Lockout_Start_Time := VI_System_Time_MS; // Блокировка на 5 минут
            END_IF;
        END_IF;
    END_IF;
    L_Prev_User_Code := VI_User_Code;

    IF L_Elapsed_Time > (GVL_CONSTANTS.C_MS_IN_MINUTE * 5) THEN
        VO_State.is_pending := FALSE; // Таймаут
    END_IF;
END_IF;

IF VO_State.Is_Locked THEN
    IF (SEL(VI_System_Time_MS >= L_Lockout_Start_Time, VI_System_Time_MS - L_Lockout_Start_Time, (4294967295 - L_Lockout_Start_Time) + VI_System_Time_MS + 1)) >= (GVL_CONSTANTS.C_MS_IN_MINUTE * 5) THEN
        VO_State.Is_Locked := FALSE;
    END_IF;
END_IF;

(* ---- FB_Ventilation_System_Manager.st ---- *)
FUNCTION_BLOCK FB_Ventilation_System_Manager
VAR_INPUT
    VI_System_Time_MS : UDINT; // Системное время (мс)
    VI_IsActivePLC : BOOL; // Флаг: Данный ПЛК является ведущим
    VI_Outdoor_Temp : REAL; // Уличная температура воздуха (°C)
    VI_Current_Scenario : E_SCENARIO_TYPE; // Текущий глобальный сценарий
    VI_System_Mode : E_System_Operating_Mode; // Агрегированный режим работы системы
    VI_Config : ST_Ventilation_Global_Config; // Конфигурация системы вентиляции
    VI_Fire_Alarm : BOOL; // Сигнал пожарной тревоги
    VI_Gas_Alarm : BOOL; // Сигнал газовой тревоги
    VI_PV3_Boost_Req : BOOL; // Запрос форсирования ПВ-3 от газоанализатора (ТЗ 5.1)
    VI_Supply_100_Req : BOOL; // Запрос 100% притока (ТЗ 6.4)
    VI_Exhaust_100_Req : BOOL; // Запрос 100% вытяжки (ТЗ 6.4)
    VI_Supply_80_Req : BOOL; // Запрос 80% притока (ТЗ 5.4)
    VI_Vent_Stop : BOOL; // Запрос на остановку вентиляции (ТЗ 5.3)
    VI_IO_Modules_Online : ARRAY[1..GVL_CONSTANTS.C_MAX_MODULES] OF BOOL; // Статусы модулей ввода-вывода (только чтение)
END_VAR
VAR_IN_OUT
    VI_Supply_Temps : ARRAY[1..GVL_CONSTANTS.C_MAX_SUPPLY_TEMPS] OF REAL; // Температура приточного воздуха после калорифера
    VI_Room_Temps : ARRAY[1..16] OF REAL; // Температура в помещениях (°C)
    VI_Room_Humidities : ARRAY[1..16] OF REAL; // Влажность в помещениях (%)
    VI_Room_CO2 : ARRAY[1..16] OF REAL; // Уровень CO2 в помещениях (ppm)
    VI_Wet_Zone_Active : ARRAY[1..GVL_CONSTANTS.C_MAX_WET_ZONES] OF BOOL; // Сигналы включения света в санузлах (ТЗ 4.0)
    VI_Rule_Actions : ARRAY[1..GVL_CONSTANTS.C_MAX_RULES] OF ST_Rule_Action; // Действия от Rule Engine
END_VAR
VAR_OUTPUT
    VO_Supply_Fans : ARRAY[1..GVL_CONSTANTS.C_MAX_SUPPLY_FANS] OF BYTE; // Выход: Управление приточными вентиляторами (0-100%)
    VO_Exhaust_Fans : ARRAY[1..GVL_CONSTANTS.C_MAX_EXHAUST_FANS] OF BYTE; // Выход: Управление вытяжными вентиляторами (0-100%)
    VO_Heater_Power : ARRAY[1..GVL_CONSTANTS.C_MAX_BOILERS] OF REAL; // Выход: Мощность калориферов (0-100%)
    VO_Status_Msg : STRING(200); // Строковое сообщение о статусе
END_VAR
VAR
    L_Policy_Normal : BOOL;
    L_Policy_Safe_Stop : BOOL;
    L_Policy_Degraded : BOOL;
    L_Policy_Freeze_Protection : BOOL;
    L_i : INT;
    L_j : INT;
    L_Max_CO2 : REAL;
    L_Max_Hum : REAL;
    L_Base_Speed : BYTE;
    L_Target_Temp : REAL;
    L_PID_Heaters : ARRAY[1..GVL_CONSTANTS.C_MAX_BOILERS] OF FB_PID_Controller;
    L_Wet_Zone_Timers : ARRAY[1..GVL_CONSTANTS.C_MAX_WET_ZONES] OF FB_System_Timer_TOF; // Таймеры выбега для вытяжек санузлов
    fbVentilationV2Staging : FB_Ventilation_V2_Staging;
    L_Vent_Command_Shadow : ST_Ventilation_Command_V2;
    L_Vent_State_Shadow : ST_Ventilation_State_V2;
    L_Vent_V2_Shadow_Diff_Found : BOOL;
    L_Vent_V2_Switch_Enabled : BOOL;
    L_Vent_V2_Path_Ready : BOOL;
    L_Vent_Using_Legacy_Fallback : BOOL;
END_VAR

// ========================================
// Ventilation policy layer (phase3/v2)
// ========================================
GVL_STATE.G_Ventilation_IO_Fault := FALSE;
GVL_STATE.G_Ventilation_Subsystem_Degraded := FALSE;
L_Vent_V2_Shadow_Diff_Found := FALSE;
L_Vent_V2_Switch_Enabled := TRUE;
L_Vent_V2_Path_Ready := FALSE;
L_Vent_Using_Legacy_Fallback := TRUE;
L_Policy_Normal := (VI_System_Mode = E_System_Operating_Mode.MODE_NORMAL);
L_Policy_Safe_Stop := (VI_System_Mode = E_System_Operating_Mode.MODE_SAFE_STOP);
L_Policy_Degraded := (VI_System_Mode = E_System_Operating_Mode.MODE_DEGRADED);
L_Policy_Freeze_Protection := (VI_System_Mode = E_System_Operating_Mode.MODE_FREEZE_PROTECTION);

IF NOT VI_IsActivePLC THEN
    FOR L_i := 1 TO GVL_CONSTANTS.C_MAX_SUPPLY_FANS DO
        VO_Supply_Fans[L_i] := 0;
        IF L_i <= GVL_CONSTANTS.C_MAX_SUPPLY_TEMPS THEN
            VO_Heater_Power[L_i] := 0.0;
        END_IF;
    END_FOR;
    FOR L_i := 1 TO GVL_CONSTANTS.C_MAX_EXHAUST_FANS DO
        VO_Exhaust_Fans[L_i] := 0;
    END_FOR;
    VO_Status_Msg := 'ВЕНТИЛЯЦИЯ: РЕЗЕРВНЫЙ ПЛК';
    RETURN;
END_IF;

// Проверка связи с модулями ввода-вывода
FOR L_i := 1 TO GVL_CONSTANTS.C_MAX_MODULES DO
    IF NOT VI_IO_Modules_Online[L_i] THEN
        GVL_STATE.G_Ventilation_IO_Fault := TRUE;
        // Переход в безопасное состояние при потере связи (отключение вентиляции)
        FOR L_j := 1 TO GVL_CONSTANTS.C_MAX_SUPPLY_FANS DO
            VO_Supply_Fans[L_j] := 0;
        END_FOR;
        FOR L_j := 1 TO GVL_CONSTANTS.C_MAX_EXHAUST_FANS DO
            VO_Exhaust_Fans[L_j] := 0;
        END_FOR;
        FOR L_j := 1 TO GVL_CONSTANTS.C_MAX_BOILERS DO
            VO_Heater_Power[L_j] := 0.0;
        END_FOR;
        VO_Status_Msg := 'ОШИБКА: Потеря связи с модулями ввода-вывода';
        RETURN;
    END_IF;
END_FOR;

// =========================
// SYSTEM MODE OVERRIDE
// =========================
// VENT_POLICY_ROUTING_PHASE3_V2
IF L_Policy_Safe_Stop THEN
    FOR L_i := 1 TO GVL_CONSTANTS.C_MAX_SUPPLY_FANS DO
        VO_Supply_Fans[L_i] := 0;
    END_FOR;
    FOR L_i := 1 TO GVL_CONSTANTS.C_MAX_EXHAUST_FANS DO
        VO_Exhaust_Fans[L_i] := 0;
    END_FOR;
    FOR L_i := 1 TO GVL_CONSTANTS.C_MAX_BOILERS DO
        VO_Heater_Power[L_i] := 0.0;
    END_FOR;
    VO_Status_Msg := 'ВЕНТИЛЯЦИЯ: ОСТАНОВЛЕНА POLICY SAFE_STOP';
    RETURN;
END_IF;

IF L_Policy_Degraded THEN
    FOR L_i := 1 TO GVL_CONSTANTS.C_MAX_SUPPLY_FANS DO
        VO_Supply_Fans[L_i] := 0;
    END_FOR;
    FOR L_i := 1 TO GVL_CONSTANTS.C_MAX_BOILERS DO
        VO_Heater_Power[L_i] := 0.0;
    END_FOR;
    GVL_STATE.G_Ventilation_Subsystem_Degraded := TRUE;
    VO_Status_Msg := 'ВЕНТИЛЯЦИЯ: DEGRADED POLICY';
END_IF;

IF L_Policy_Freeze_Protection THEN
    FOR L_i := 1 TO GVL_CONSTANTS.C_MAX_SUPPLY_FANS DO
        VO_Supply_Fans[L_i] := 0;
    END_FOR;
    FOR L_i := 1 TO GVL_CONSTANTS.C_MAX_EXHAUST_FANS DO
        VO_Exhaust_Fans[L_i] := 0;
    END_FOR;
    FOR L_i := 1 TO GVL_CONSTANTS.C_MAX_BOILERS DO
        VO_Heater_Power[L_i] := 0.0;
    END_FOR;
    VO_Status_Msg := 'ВЕНТИЛЯЦИЯ: FREEZE_PROTECTION POLICY (stop)';
    RETURN;
END_IF;

// MODE_FREEZE_PROTECTION пока оставляем на текущей штатной логике

// 1. Определение базовой скорости и целевой температуры по сценарию (ТЗ 7.1)
CASE VI_Current_Scenario OF
    E_SCENARIO_TYPE.SCENARIO_AWAY:
        L_Base_Speed := VI_Config.Scenario_Modes[3].Base_Fan_Speed;
        L_Target_Temp := VI_Config.Scenario_Modes[3].Target_Temp;
    E_SCENARIO_TYPE.SCENARIO_SLEEP:
        L_Base_Speed := VI_Config.Scenario_Modes[2].Base_Fan_Speed;
        L_Target_Temp := VI_Config.Scenario_Modes[2].Target_Temp;
    ELSE // PRESENCE, MORNING, EVENING
        L_Base_Speed := VI_Config.Scenario_Modes[1].Base_Fan_Speed;
        L_Target_Temp := VI_Config.Scenario_Modes[1].Target_Temp;
END_CASE;

// 2. Логика управления приточными установками (П-1, П-2, П-3)
FOR L_i := 1 TO GVL_CONSTANTS.C_MAX_SUPPLY_FANS DO
    // ПИД-регулирование мощности электрического калорифера
    IF L_i <= GVL_CONSTANTS.C_MAX_SUPPLY_TEMPS THEN
        L_PID_Heaters[L_i](
            VI_SetPoint := L_Target_Temp,
            VI_ProcessValue := VI_Supply_Temps[L_i], // Используем датчик температуры после калорифера
            VI_Kp := 4.0, VI_Tn := 120.0, VI_Tv := 0.0,
            VI_Y_Min := 0.0, VI_Y_Max := 100.0, VI_Cycle_Time_S := 1.0,
            VO_Output => VO_Heater_Power[L_i]
        );
    END_IF;

    // Определение скорости приточного вентилятора
    VO_Supply_Fans[L_i] := L_Base_Speed;

    // Обработка действий от Rule Engine
    FOR L_j := 1 TO GVL_CONSTANTS.C_MAX_RULES DO
        IF VI_Rule_Actions[L_j].Active AND VI_Rule_Actions[L_j].Target_ID = L_i THEN
            IF VI_Rule_Actions[L_j].Action_Type = E_Rule_Action_Type.ACTION_SET_VENTILATION THEN
                VO_Supply_Fans[L_i] := REAL_TO_BYTE(VI_Rule_Actions[L_j].Value);
            END_IF;
        END_IF;
    END_FOR;

    // Requests are observed but must not bypass policy directly.
    IF VI_Supply_100_Req OR VI_Supply_80_Req OR VI_Fire_Alarm OR VI_Vent_Stop OR VI_Gas_Alarm OR VI_PV3_Boost_Req THEN
        GVL_STATE.G_Ventilation_Subsystem_Degraded := TRUE;
    END_IF;
END_FOR;

// 3. Логика управления вытяжными установками (В-1 .. В-5)
FOR L_i := 1 TO GVL_CONSTANTS.C_MAX_EXHAUST_FANS DO
    VO_Exhaust_Fans[L_i] := L_Base_Speed;

    // ТЗ 4.0: Логика вытяжки в санузлах
    FOR L_j := 1 TO GVL_CONSTANTS.C_MAX_WET_ZONES DO
        IF VI_Config.wet_zone_to_exhaust_map[L_j] = L_i THEN
            // Включение по свету, выключение с задержкой 5 минут (используем TOF)
            L_Wet_Zone_Timers[L_j](IN := VI_Wet_Zone_Active[L_j], PT := T#5m, VI_System_Time_MS := VI_System_Time_MS);
            IF VI_Wet_Zone_Active[L_j] THEN
                VO_Exhaust_Fans[L_i] := 80; // Повышенная скорость при присутствии
            ELSIF L_Wet_Zone_Timers[L_j].Q THEN
                VO_Exhaust_Fans[L_i] := 50; // Скорость выбега (пока таймер TOF активен)
            END_IF;
        END_IF;
    END_FOR;

    // Requests are observed but must not bypass policy directly.
    IF (L_i = VI_Config.pv3_exhaust_index AND VI_PV3_Boost_Req) OR VI_Exhaust_100_Req OR VI_Fire_Alarm OR VI_Vent_Stop OR VI_Gas_Alarm THEN
        GVL_STATE.G_Ventilation_Subsystem_Degraded := TRUE;
    END_IF;
END_FOR;

// ========================================
// VENT_FINAL_CLAMP
// ========================================
IF L_Policy_Degraded THEN
    FOR L_i := 1 TO GVL_CONSTANTS.C_MAX_EXHAUST_FANS DO
        VO_Exhaust_Fans[L_i] := MIN(VO_Exhaust_Fans[L_i], VI_Config.Degraded_Exhaust_Limit);
    END_FOR;
END_IF;

// Ventilation V2 shadow runtime integration (diagnostic only)
fbVentilationV2Staging(
    VI_Zone_ID := 1,
    VI_Enable := (NOT L_Policy_Safe_Stop) AND (NOT L_Policy_Freeze_Protection) AND (NOT GVL_STATE.G_Ventilation_IO_Fault),
    VI_Fan_Speed_Setpoint := BYTE_TO_REAL(VO_Supply_Fans[1]),
    VI_Damper_Position_Setpoint := 0.0,
    VI_Heat_Recovery_Enabled := L_Policy_Normal,
    VI_Is_Active := (VO_Supply_Fans[1] > 0) OR (VO_Exhaust_Fans[1] > 0),
    VI_Fan_Speed_Actual := BYTE_TO_REAL(VO_Supply_Fans[1]),
    VI_Supply_Temp := VI_Supply_Temps[1],
    VI_Extract_Temp := VI_Room_Temps[1],
    VI_Filter_Dirty := FALSE,
    VI_Alarm_Active := GVL_STATE.G_Ventilation_IO_Fault OR GVL_STATE.G_Ventilation_Subsystem_Degraded,
    VO_Command_Shadow => L_Vent_Command_Shadow,
    VO_State_Shadow => L_Vent_State_Shadow
);

// Ventilation V2 shadow validation
IF ABS(BYTE_TO_REAL(VO_Supply_Fans[1]) - L_Vent_Command_Shadow.Fan_Speed_Setpoint) > 0.1 THEN
    L_Vent_V2_Shadow_Diff_Found := TRUE;
END_IF;
IF ABS(VI_Supply_Temps[1] - L_Vent_State_Shadow.Supply_Temp) > 0.1 THEN
    L_Vent_V2_Shadow_Diff_Found := TRUE;
END_IF;

// Guarded Ventilation V2 enable
IF L_Vent_V2_Switch_Enabled THEN
    IF NOT L_Vent_V2_Shadow_Diff_Found THEN
        L_Vent_V2_Path_Ready := TRUE;
        L_Vent_Using_Legacy_Fallback := FALSE;
    ELSE
        L_Vent_V2_Path_Ready := FALSE;
        L_Vent_Using_Legacy_Fallback := TRUE;
    END_IF;
ELSE
    L_Vent_V2_Path_Ready := FALSE;
    L_Vent_Using_Legacy_Fallback := TRUE;
END_IF;

// 4. Формирование статусного сообщения
IF L_Policy_Safe_Stop THEN
    VO_Status_Msg := 'ВЕНТИЛЯЦИЯ: ОСТАНОВЛЕНА POLICY SAFE_STOP';
ELSIF L_Policy_Freeze_Protection THEN
    VO_Status_Msg := 'ВЕНТИЛЯЦИЯ: FREEZE_PROTECTION POLICY (stop)';
ELSIF L_Policy_Degraded THEN
    VO_Status_Msg := 'ВЕНТИЛЯЦИЯ: DEGRADED POLICY';
ELSE
    VO_Status_Msg := 'Вентиляция работает в штатном режиме';
END_IF;
// >>> BULK_SYNC_ANCHOR: FB_Ventilation_System_Manager <<<

(* ---- FB_Ventilation_V2_Staging.st ---- *)
FUNCTION_BLOCK FB_Ventilation_V2_Staging
VAR_INPUT
    VI_Zone_ID : INT;
    VI_Enable : BOOL;
    VI_Fan_Speed_Setpoint : REAL;
    VI_Damper_Position_Setpoint : REAL;
    VI_Heat_Recovery_Enabled : BOOL;
    VI_Is_Active : BOOL;
    VI_Fan_Speed_Actual : REAL;
    VI_Supply_Temp : REAL;
    VI_Extract_Temp : REAL;
    VI_Filter_Dirty : BOOL;
    VI_Alarm_Active : BOOL;
END_VAR
VAR_OUTPUT
    VO_Command_Shadow : ST_Ventilation_Command_V2;
    VO_State_Shadow : ST_Ventilation_State_V2;
END_VAR

VO_Command_Shadow.Fan_Speed_Setpoint := VI_Fan_Speed_Setpoint;
VO_State_Shadow.Supply_Temp := VI_Supply_Temp;
END_FUNCTION_BLOCK

(* ---- MAIN.st ---- *)
PROGRAM MAIN
VAR
END_VAR

// Вызов основных программ
PRG_IO_Read();
PRG_System();
PRG_Safety();
PRG_Security();
PRG_Heating();
PRG_Ventilation();
PRG_Lighting();
PRG_IO_Write();

// PRG_Test(); // Раскомментировать для запуска модульных тестов

(* ---- PRG_PLC_A.st ---- *)
PROGRAM PRG_PLC_A
VAR
    // Специфичная логика для ПЛК А
END_VAR

// Вызов основной программы
PRG_System();
// >>> BULK_SYNC_ANCHOR: PRG_PLC_A <<<

(* ---- PRG_PLC_B.st ---- *)
PROGRAM PRG_PLC_B
VAR
    // Специфичная логика для ПЛК B
END_VAR

// Вызов основной программы
PRG_System();
// >>> BULK_SYNC_ANCHOR: PRG_PLC_B <<<
